// Nodes/Algebraic Container Ops/AddTo/Node_F_VN_AddToContainerElements_TcVnVector4_UINT
{attribute 'linkalways'} 
{attribute 'no_explicit_call' := 'This FB is a CLASS and must be accessed using methods or properties'}
{attribute 'enable_dynamic_creation'}
FUNCTION_BLOCK Node_F_VN_AddToContainerElements_TcVnVector4_UINT EXTENDS VisionNode
VAR
    aValue : _TcVnVector4_UINT;
    ipContainer : _ITcVnContainer;
    hrPrev : _HRESULT(S_OK);
    hresult : _HRESULT(S_OK);
END_VAR

METHOD FB_init : BOOL
VAR_INPUT
    bInitRetains : BOOL; // if TRUE, the retain variables are initialized (warm start / cold start)
    bInCopyCode : BOOL;  // if TRUE, the instance afterwards gets moved into the copy code (online change)
END_VAR
AddInput('aValue', aValue);
AddInput('ipContainer', ipContainer);
AddInput('hrPrev', hrPrev);
AddOutput('ipContainer', ipContainer);
AddOutput('hresult',hresult);
END_METHOD

METHOD PUBLIC  Clone : I_Node
VAR
    pNode : POINTER TO Node_F_VN_AddToContainerElements_TcVnVector4_UINT;
END_VAR
pNode := __NEW(Node_F_VN_AddToContainerElements_TcVnVector4_UINT);
Clone := pNode^;
END_METHOD

METHOD PROTECTED OnExecute
hresult.Value := F_VN_AddToContainerElements_TcVnVector4_UINT(
    aValue := aValue.Value,
    ipContainer := ipContainer.Value,
    hrPrev:= hrPrev.Value);
END_METHOD

METHOD PUBLIC PreExecutionCheck
VAR_INPUT
    Check : I_PreExecutionChecks;
END_VAR
Check.IsTrue(ipContainer.IsValid, 'ipContainer must be a valid container');
Check.IsTrue(ipContainer.IsType(TC_GLOBAL_CONST_LIST.ContainerType_Vector_TcVnVector4_UINT), 'ipContainer contains incorrect type');
END_METHOD

END_FUNCTION_BLOCK

// Nodes/Algebraic Container Ops/AddTo/Node_F_VN_AddToContainerElements_TcVnVector4_USINT
{attribute 'linkalways'} 
{attribute 'no_explicit_call' := 'This FB is a CLASS and must be accessed using methods or properties'}
{attribute 'enable_dynamic_creation'}
FUNCTION_BLOCK Node_F_VN_AddToContainerElements_TcVnVector4_USINT EXTENDS VisionNode
VAR
    aValue : _TcVnVector4_USINT;
    ipContainer : _ITcVnContainer;
    hrPrev : _HRESULT(S_OK);
    hresult : _HRESULT(S_OK);
END_VAR

METHOD FB_init : BOOL
VAR_INPUT
    bInitRetains : BOOL; // if TRUE, the retain variables are initialized (warm start / cold start)
    bInCopyCode : BOOL;  // if TRUE, the instance afterwards gets moved into the copy code (online change)
END_VAR
AddInput('aValue', aValue);
AddInput('ipContainer', ipContainer);
AddInput('hrPrev', hrPrev);
AddOutput('ipContainer', ipContainer);
AddOutput('hresult',hresult);
END_METHOD

METHOD PUBLIC  Clone : I_Node
VAR
    pNode : POINTER TO Node_F_VN_AddToContainerElements_TcVnVector4_USINT;
END_VAR
pNode := __NEW(Node_F_VN_AddToContainerElements_TcVnVector4_USINT);
Clone := pNode^;
END_METHOD

METHOD PROTECTED OnExecute
hresult.Value := F_VN_AddToContainerElements_TcVnVector4_USINT(
    aValue := aValue.Value,
    ipContainer := ipContainer.Value,
    hrPrev:= hrPrev.Value);
END_METHOD

METHOD PUBLIC PreExecutionCheck
VAR_INPUT
    Check : I_PreExecutionChecks;
END_VAR
Check.IsTrue(ipContainer.IsValid, 'ipContainer must be a valid container');
Check.IsTrue(ipContainer.IsType(TC_GLOBAL_CONST_LIST.ContainerType_Vector_TcVnVector4_USINT), 'ipContainer contains incorrect type');
END_METHOD

END_FUNCTION_BLOCK

// Nodes/Algebraic Container Ops/AddTo/Node_F_VN_AddToContainerElements_UDINT
{attribute 'linkalways'} 
{attribute 'no_explicit_call' := 'This FB is a CLASS and must be accessed using methods or properties'}
{attribute 'enable_dynamic_creation'}
FUNCTION_BLOCK Node_F_VN_AddToContainerElements_UDINT EXTENDS VisionNode
VAR
    nValue : _UDINT(0);
    ipContainer : _ITcVnContainer;
    hrPrev : _HRESULT(S_OK);
    hresult : _HRESULT(S_OK);
END_VAR

METHOD FB_init : BOOL
VAR_INPUT
    bInitRetains : BOOL; // if TRUE, the retain variables are initialized (warm start / cold start)
    bInCopyCode : BOOL;  // if TRUE, the instance afterwards gets moved into the copy code (online change)
END_VAR
AddParameter('nValue', nValue);
AddInput('ipContainer', ipContainer);
AddInput('hrPrev', hrPrev);
AddOutput('ipContainer', ipContainer);
AddOutput('hresult',hresult);
END_METHOD

METHOD PUBLIC  Clone : I_Node
VAR
    pNode : POINTER TO Node_F_VN_AddToContainerElements_UDINT;
END_VAR
pNode := __NEW(Node_F_VN_AddToContainerElements_UDINT);
Clone := pNode^;
END_METHOD

METHOD PROTECTED OnExecute
hresult.Value := F_VN_AddToContainerElements_UDINT(
    nValue := nValue.Value,
    ipContainer := ipContainer.Value,
    hrPrev:= hrPrev.Value);
END_METHOD

METHOD PUBLIC PreExecutionCheck
VAR_INPUT
    Check : I_PreExecutionChecks;
END_VAR
Check.IsTrue(ipContainer.IsValid, 'ipContainer must be a valid container');
Check.IsTrue(ipContainer.IsType(TC_GLOBAL_CONST_LIST.ContainerType_Vector_UDINT), 'ipContainer contains incorrect type');
END_METHOD

END_FUNCTION_BLOCK

// Nodes/Algebraic Container Ops/AddTo/Node_F_VN_AddToContainerElements_UINT
{attribute 'linkalways'} 
{attribute 'no_explicit_call' := 'This FB is a CLASS and must be accessed using methods or properties'}
{attribute 'enable_dynamic_creation'}
FUNCTION_BLOCK Node_F_VN_AddToContainerElements_UINT EXTENDS VisionNode
VAR
    nValue : _UINT(0);
    ipContainer : _ITcVnContainer;
    hrPrev : _HRESULT(S_OK);
    hresult : _HRESULT(S_OK);
END_VAR

METHOD FB_init : BOOL
VAR_INPUT
    bInitRetains : BOOL; // if TRUE, the retain variables are initialized (warm start / cold start)
    bInCopyCode : BOOL;  // if TRUE, the instance afterwards gets moved into the copy code (online change)
END_VAR
AddParameter('nValue', nValue);
AddInput('ipContainer', ipContainer);
AddInput('hrPrev', hrPrev);
AddOutput('ipContainer', ipContainer);
AddOutput('hresult',hresult);
END_METHOD

METHOD PUBLIC  Clone : I_Node
VAR
    pNode : POINTER TO Node_F_VN_AddToContainerElements_UINT;
END_VAR
pNode := __NEW(Node_F_VN_AddToContainerElements_UINT);
Clone := pNode^;
END_METHOD

METHOD PROTECTED OnExecute
hresult.Value := F_VN_AddToContainerElements_UINT(
    nValue := nValue.Value,
    ipContainer := ipContainer.Value,
    hrPrev:= hrPrev.Value);
END_METHOD

METHOD PUBLIC PreExecutionCheck
VAR_INPUT
    Check : I_PreExecutionChecks;
END_VAR
Check.IsTrue(ipContainer.IsValid, 'ipContainer must be a valid container');
Check.IsTrue(ipContainer.IsType(TC_GLOBAL_CONST_LIST.ContainerType_Vector_UINT), 'ipContainer contains incorrect type');
END_METHOD

END_FUNCTION_BLOCK

// Nodes/Algebraic Container Ops/AddTo/Node_F_VN_AddToContainerElements_ULINT
{attribute 'linkalways'} 
{attribute 'no_explicit_call' := 'This FB is a CLASS and must be accessed using methods or properties'}
{attribute 'enable_dynamic_creation'}
FUNCTION_BLOCK Node_F_VN_AddToContainerElements_ULINT EXTENDS VisionNode
VAR
    nValue : _ULINT(0);
    ipContainer : _ITcVnContainer;
    hrPrev : _HRESULT(S_OK);
    hresult : _HRESULT(S_OK);
END_VAR

METHOD FB_init : BOOL
VAR_INPUT
    bInitRetains : BOOL; // if TRUE, the retain variables are initialized (warm start / cold start)
    bInCopyCode : BOOL;  // if TRUE, the instance afterwards gets moved into the copy code (online change)
END_VAR
AddParameter('nValue', nValue);
AddInput('ipContainer', ipContainer);
AddInput('hrPrev', hrPrev);
AddOutput('ipContainer', ipContainer);
AddOutput('hresult',hresult);
END_METHOD

METHOD PUBLIC  Clone : I_Node
VAR
    pNode : POINTER TO Node_F_VN_AddToContainerElements_ULINT;
END_VAR
pNode := __NEW(Node_F_VN_AddToContainerElements_ULINT);
Clone := pNode^;
END_METHOD

METHOD PROTECTED OnExecute
hresult.Value := F_VN_AddToContainerElements_ULINT(
    nValue := nValue.Value,
    ipContainer := ipContainer.Value,
    hrPrev:= hrPrev.Value);
END_METHOD

METHOD PUBLIC PreExecutionCheck
VAR_INPUT
    Check : I_PreExecutionChecks;
END_VAR
Check.IsTrue(ipContainer.IsValid, 'ipContainer must be a valid container');
Check.IsTrue(ipContainer.IsType(TC_GLOBAL_CONST_LIST.ContainerType_Vector_ULINT), 'ipContainer contains incorrect type');
END_METHOD

END_FUNCTION_BLOCK

// Nodes/Algebraic Container Ops/AddTo/Node_F_VN_AddToContainerElements_USINT
{attribute 'linkalways'} 
{attribute 'no_explicit_call' := 'This FB is a CLASS and must be accessed using methods or properties'}
{attribute 'enable_dynamic_creation'}
FUNCTION_BLOCK Node_F_VN_AddToContainerElements_USINT EXTENDS VisionNode
VAR
    nValue : _USINT(0);
    ipContainer : _ITcVnContainer;
    hrPrev : _HRESULT(S_OK);
    hresult : _HRESULT(S_OK);
END_VAR

METHOD FB_init : BOOL
VAR_INPUT
    bInitRetains : BOOL; // if TRUE, the retain variables are initialized (warm start / cold start)
    bInCopyCode : BOOL;  // if TRUE, the instance afterwards gets moved into the copy code (online change)
END_VAR
AddParameter('nValue', nValue);
AddInput('ipContainer', ipContainer);
AddInput('hrPrev', hrPrev);
AddOutput('ipContainer', ipContainer);
AddOutput('hresult',hresult);
END_METHOD

METHOD PUBLIC  Clone : I_Node
VAR
    pNode : POINTER TO Node_F_VN_AddToContainerElements_USINT;
END_VAR
pNode := __NEW(Node_F_VN_AddToContainerElements_USINT);
Clone := pNode^;
END_METHOD

METHOD PROTECTED OnExecute
hresult.Value := F_VN_AddToContainerElements_USINT(
    nValue := nValue.Value,
    ipContainer := ipContainer.Value,
    hrPrev:= hrPrev.Value);
END_METHOD

METHOD PUBLIC PreExecutionCheck
VAR_INPUT
    Check : I_PreExecutionChecks;
END_VAR
Check.IsTrue(ipContainer.IsValid, 'ipContainer must be a valid container');
Check.IsTrue(ipContainer.IsType(TC_GLOBAL_CONST_LIST.ContainerType_Vector_USINT), 'ipContainer contains incorrect type');
END_METHOD

END_FUNCTION_BLOCK

// Nodes/Algebraic Container Ops/Node_F_VN_AddContainers
{attribute 'linkalways'} 
{attribute 'no_explicit_call' := 'This FB is a CLASS and must be accessed using methods or properties'}
{attribute 'enable_dynamic_creation'}
FUNCTION_BLOCK Node_F_VN_AddContainers EXTENDS VisionNode
VAR
    ipSrcContainer1 : _ITcVnContainer;
    ipSrcContainer2 : _ITcVnContainer;
    ipDestContainer : _ITcVnContainer;
    hrPrev : _HRESULT(S_OK);
    hresult : _HRESULT(S_OK);
END_VAR

METHOD FB_init : BOOL
VAR_INPUT
    bInitRetains : BOOL; // if TRUE, the retain variables are initialized (warm start / cold start)
    bInCopyCode : BOOL;  // if TRUE, the instance afterwards gets moved into the copy code (online change)
END_VAR
AddInput('ipSrcContainer1', ipSrcContainer1);
AddInput('ipSrcContainer2', ipSrcContainer2);
AddInput('hrPrev', hrPrev);
AddOutput('ipDestContainer', ipDestContainer);
AddOutput('hresult',hresult);
END_METHOD

METHOD PUBLIC  Clone : I_Node
VAR
    pNode : POINTER TO Node_F_VN_AddContainers;
END_VAR
pNode := __NEW(Node_F_VN_AddContainers);
Clone := pNode^;
END_METHOD

METHOD PROTECTED OnExecute
hresult.Value := F_VN_AddContainers(
    ipSrcContainer1 := ipSrcContainer1.Value,
    ipSrcContainer2 := ipSrcContainer2.Value,
    ipDestContainer := ipDestContainer.Value,
    hrPrev:= hrPrev.Value);
END_METHOD

METHOD PUBLIC PreExecutionCheck
VAR_INPUT
    Check : I_PreExecutionChecks;
END_VAR
Check.IsTrue(ipSrcContainer1.IsValid, 'ipSrcContainer1 must be a valid container');
Check.IsTrue(ipSrcContainer2.IsValid, 'ipSrcContainer2 must be a valid container');
Check.IsTrue(ContainersHaveMatchingTypes(ipSrcContainer1.Value, ipSrcContainer2.Value), 'Source containers must have matching types');
Check.IsTrue(ContainersHaveMatchingNumberOfElements(ipSrcContainer1.Value, ipSrcContainer2.Value), 'Source containers must contain the same number of elements');
END_METHOD

END_FUNCTION_BLOCK

// Nodes/Algebraic Container Ops/Node_F_VN_BitwiseAndContainers
{attribute 'linkalways'} 
{attribute 'no_explicit_call' := 'This FB is a CLASS and must be accessed using methods or properties'}
{attribute 'enable_dynamic_creation'}
FUNCTION_BLOCK Node_F_VN_BitwiseAndContainers EXTENDS VisionNode
VAR
    ipSrcContainer1 : _ITcVnContainer;
    ipSrcContainer2 : _ITcVnContainer;
    ipDestContainer : _ITcVnContainer;
    hrPrev : _HRESULT(S_OK);
    hresult : _HRESULT(S_OK);
END_VAR

METHOD FB_init : BOOL
VAR_INPUT
    bInitRetains : BOOL; // if TRUE, the retain variables are initialized (warm start / cold start)
    bInCopyCode : BOOL;  // if TRUE, the instance afterwards gets moved into the copy code (online change)
END_VAR
AddInput('ipSrcContainer1', ipSrcContainer1);
AddInput('ipSrcContainer2', ipSrcContainer2);
AddInput('hrPrev', hrPrev);
AddOutput('ipDestContainer', ipDestContainer);
AddOutput('hresult',hresult);
END_METHOD

METHOD PUBLIC  Clone : I_Node
VAR
    pNode : POINTER TO Node_F_VN_BitwiseAndContainers;
END_VAR
pNode := __NEW(Node_F_VN_BitwiseAndContainers);
Clone := pNode^;
END_METHOD

METHOD PROTECTED OnExecute
hresult.Value := F_VN_BitwiseAndContainers(
    ipSrcContainer1 := ipSrcContainer1.Value,
    ipSrcContainer2 := ipSrcContainer2.Value,
    ipDestContainer := ipDestContainer.Value,
    hrPrev:= hrPrev.Value);
END_METHOD

METHOD PUBLIC PreExecutionCheck
VAR_INPUT
    Check : I_PreExecutionChecks;
END_VAR
Check.IsTrue(ipSrcContainer1.IsValid, 'ipSrcContainer1 must be a valid container');
Check.IsTrue(ipSrcContainer2.IsValid, 'ipSrcContainer2 must be a valid container');
Check.IsTrue(ContainersHaveMatchingTypes(ipSrcContainer1.Value, ipSrcContainer2.Value), 'Source containers must have matching types');
Check.IsTrue(ContainersHaveMatchingNumberOfElements(ipSrcContainer1.Value, ipSrcContainer2.Value), 'Source containers must contain the same number of elements');


//TODO Need to check that container has integer values only.
// SINT, USINT, INT, UINT, DINT, UDINT, ULINT only?
END_METHOD

END_FUNCTION_BLOCK

// Nodes/Algebraic Container Ops/Node_F_VN_BitwiseNotContainer
{attribute 'linkalways'} 
{attribute 'no_explicit_call' := 'This FB is a CLASS and must be accessed using methods or properties'}
{attribute 'enable_dynamic_creation'}
FUNCTION_BLOCK Node_F_VN_BitwiseNotContainer EXTENDS VisionNode
VAR
    ipSrcContainer : _ITcVnContainer;
    ipDestContainer : _ITcVnContainer;
    hrPrev : _HRESULT(S_OK);
    hresult : _HRESULT(S_OK);
END_VAR

METHOD FB_init : BOOL
VAR_INPUT
    bInitRetains : BOOL; // if TRUE, the retain variables are initialized (warm start / cold start)
    bInCopyCode : BOOL;  // if TRUE, the instance afterwards gets moved into the copy code (online change)
END_VAR
AddInput('ipSrcContainer', ipSrcContainer);
AddInput('hrPrev', hrPrev);
AddOutput('ipDestContainer', ipDestContainer);
AddOutput('hresult',hresult);
END_METHOD

METHOD PUBLIC  Clone : I_Node
VAR
    pNode : POINTER TO Node_F_VN_BitwiseNotContainer;
END_VAR
pNode := __NEW(Node_F_VN_BitwiseNotContainer);
Clone := pNode^;
END_METHOD

METHOD PROTECTED OnExecute
hresult.Value := F_VN_BitwiseNotContainer(
    ipSrcContainer := ipSrcContainer.Value,
    ipDestContainer := ipDestContainer.Value,
    hrPrev:= hrPrev.Value);
END_METHOD

METHOD PUBLIC PreExecutionCheck
VAR_INPUT
    Check : I_PreExecutionChecks;
END_VAR
Check.IsTrue(ipSrcContainer.IsValid, 'ipSrcContainer must be a valid container');

IF Check.Failed THEN
    RETURN;
END_IF

//TODO Need to check that container has integer values only.
// SINT, USINT, INT, UINT, DINT, UDINT, ULINT only?
END_METHOD

END_FUNCTION_BLOCK

// Nodes/Algebraic Container Ops/Node_F_VN_BitwiseOrContainers
{attribute 'linkalways'} 
{attribute 'no_explicit_call' := 'This FB is a CLASS and must be accessed using methods or properties'}
{attribute 'enable_dynamic_creation'}
FUNCTION_BLOCK Node_F_VN_BitwiseOrContainers EXTENDS VisionNode
VAR
    ipSrcContainer1 : _ITcVnContainer;
    ipSrcContainer2 : _ITcVnContainer;
    ipDestContainer : _ITcVnContainer;
    hrPrev : _HRESULT(S_OK);
    hresult : _HRESULT(S_OK);
END_VAR

METHOD FB_init : BOOL
VAR_INPUT
    bInitRetains : BOOL; // if TRUE, the retain variables are initialized (warm start / cold start)
    bInCopyCode : BOOL;  // if TRUE, the instance afterwards gets moved into the copy code (online change)
END_VAR
AddInput('ipSrcContainer1', ipSrcContainer1);
AddInput('ipSrcContainer2', ipSrcContainer2);
AddInput('hrPrev', hrPrev);
AddOutput('ipDestContainer', ipDestContainer);
AddOutput('hresult',hresult);
END_METHOD

METHOD PUBLIC  Clone : I_Node
VAR
    pNode : POINTER TO Node_F_VN_BitwiseOrContainers;
END_VAR
pNode := __NEW(Node_F_VN_BitwiseOrContainers);
Clone := pNode^;
END_METHOD

METHOD PROTECTED OnExecute
hresult.Value := F_VN_BitwiseOrContainers(
    ipSrcContainer1 := ipSrcContainer1.Value,
    ipSrcContainer2 := ipSrcContainer2.Value,
    ipDestContainer := ipDestContainer.Value,
    hrPrev:= hrPrev.Value);
END_METHOD

METHOD PUBLIC PreExecutionCheck
VAR_INPUT
    Check : I_PreExecutionChecks;
END_VAR
Check.IsTrue(ipSrcContainer1.IsValid, 'ipSrcContainer1 must be a valid container');
Check.IsTrue(ipSrcContainer2.IsValid, 'ipSrcContainer2 must be a valid container');
Check.IsTrue(ContainersHaveMatchingTypes(ipSrcContainer1.Value, ipSrcContainer2.Value), 'Source containers must have matching types');
Check.IsTrue(ContainersHaveMatchingNumberOfElements(ipSrcContainer1.Value, ipSrcContainer2.Value), 'Source containers must contain the same number of elements');


//TODO Need to check that container has integer values only.
// SINT, USINT, INT, UINT, DINT, UDINT, ULINT only?
END_METHOD

END_FUNCTION_BLOCK

// Nodes/Algebraic Container Ops/Node_F_VN_BitwiseXorContainers
{attribute 'linkalways'} 
{attribute 'no_explicit_call' := 'This FB is a CLASS and must be accessed using methods or properties'}
{attribute 'enable_dynamic_creation'}
FUNCTION_BLOCK Node_F_VN_BitwiseXorContainers EXTENDS VisionNode
VAR
    ipSrcContainer1 : _ITcVnContainer;
    ipSrcContainer2 : _ITcVnContainer;
    ipDestContainer : _ITcVnContainer;
    hrPrev : _HRESULT(S_OK);
    hresult : _HRESULT(S_OK);
END_VAR

METHOD FB_init : BOOL
VAR_INPUT
    bInitRetains : BOOL; // if TRUE, the retain variables are initialized (warm start / cold start)
    bInCopyCode : BOOL;  // if TRUE, the instance afterwards gets moved into the copy code (online change)
END_VAR
AddInput('ipSrcContainer1', ipSrcContainer1);
AddInput('ipSrcContainer2', ipSrcContainer2);
AddInput('hrPrev', hrPrev);
AddOutput('ipDestContainer', ipDestContainer);
AddOutput('hresult',hresult);
END_METHOD

METHOD PUBLIC  Clone : I_Node
VAR
    pNode : POINTER TO Node_F_VN_BitwiseXorContainers;
END_VAR
pNode := __NEW(Node_F_VN_BitwiseXorContainers);
Clone := pNode^;
END_METHOD

METHOD PROTECTED OnExecute
hresult.Value := F_VN_BitwiseXorContainers(
    ipSrcContainer1 := ipSrcContainer1.Value,
    ipSrcContainer2 := ipSrcContainer2.Value,
    ipDestContainer := ipDestContainer.Value,
    hrPrev:= hrPrev.Value);
END_METHOD

METHOD PUBLIC PreExecutionCheck
VAR_INPUT
    Check : I_PreExecutionChecks;
END_VAR
Check.IsTrue(ipSrcContainer1.IsValid, 'ipSrcContainer1 must be a valid container');
Check.IsTrue(ipSrcContainer2.IsValid, 'ipSrcContainer2 must be a valid container');
Check.IsTrue(ContainersHaveMatchingTypes(ipSrcContainer1.Value, ipSrcContainer2.Value), 'Source containers must have matching types');
Check.IsTrue(ContainersHaveMatchingNumberOfElements(ipSrcContainer1.Value, ipSrcContainer2.Value), 'Source containers must contain the same number of elements');

//TODO Need to check that container has integer values only.
// SINT, USINT, INT, UINT, DINT, UDINT, ULINT only?
END_METHOD

END_FUNCTION_BLOCK

// Nodes/Algebraic Container Ops/Node_F_VN_DivideContainers
{attribute 'linkalways'} 
{attribute 'no_explicit_call' := 'This FB is a CLASS and must be accessed using methods or properties'}
{attribute 'enable_dynamic_creation'}
FUNCTION_BLOCK Node_F_VN_DivideContainers EXTENDS VisionNode
VAR
    ipSrcContainer1 : _ITcVnContainer;
    ipSrcContainer2 : _ITcVnContainer;
    ipDestContainer : _ITcVnContainer;
    hrPrev : _HRESULT(S_OK);
    hresult : _HRESULT(S_OK);
END_VAR

METHOD FB_init : BOOL
VAR_INPUT
    bInitRetains : BOOL; // if TRUE, the retain variables are initialized (warm start / cold start)
    bInCopyCode : BOOL;  // if TRUE, the instance afterwards gets moved into the copy code (online change)
END_VAR
AddInput('ipSrcContainer1', ipSrcContainer1);
AddInput('ipSrcContainer2', ipSrcContainer2);
AddInput('hrPrev', hrPrev);
AddOutput('ipDestContainer', ipDestContainer);
AddOutput('hresult',hresult);
END_METHOD

METHOD PUBLIC  Clone : I_Node
VAR
    pNode : POINTER TO Node_F_VN_DivideContainers;
END_VAR
pNode := __NEW(Node_F_VN_DivideContainers);
Clone := pNode^;
END_METHOD

METHOD PROTECTED OnExecute
hresult.Value := F_VN_DivideContainers(
    ipSrcContainer1 := ipSrcContainer1.Value,
    ipSrcContainer2 := ipSrcContainer2.Value,
    ipDestContainer := ipDestContainer.Value,
    hrPrev:= hrPrev.Value);
END_METHOD

METHOD PUBLIC PreExecutionCheck
VAR_INPUT
    Check : I_PreExecutionChecks;
END_VAR
Check.IsTrue(ipSrcContainer1.IsValid, 'ipSrcContainer1 must be a valid container');
Check.IsTrue(ipSrcContainer2.IsValid, 'ipSrcContainer2 must be a valid container');
Check.IsTrue(ContainersHaveMatchingTypes(ipSrcContainer1.Value, ipSrcContainer2.Value), 'Source containers must have matching types');
Check.IsTrue(ContainersHaveMatchingNumberOfElements(ipSrcContainer1.Value, ipSrcContainer2.Value), 'Source containers must contain the same number of elements');
END_METHOD

END_FUNCTION_BLOCK

// Nodes/Algebraic Container Ops/Node_F_VN_DivideContainersExp
{attribute 'linkalways'} 
{attribute 'no_explicit_call' := 'This FB is a CLASS and must be accessed using methods or properties'}
{attribute 'enable_dynamic_creation'}
FUNCTION_BLOCK Node_F_VN_DivideContainersExp EXTENDS VisionNode
VAR
    ipSrcContainer1 : _ITcVnContainer;
    ipSrcContainer2 : _ITcVnContainer;
    ipDestContainer : _ITcVnContainer;
    nIntDivideByZeroResult : _LINT(0);
    hrPrev : _HRESULT(S_OK);
    hresult : _HRESULT(S_OK);
END_VAR

METHOD FB_init : BOOL
VAR_INPUT
    bInitRetains : BOOL; // if TRUE, the retain variables are initialized (warm start / cold start)
    bInCopyCode : BOOL;  // if TRUE, the instance afterwards gets moved into the copy code (online change)
END_VAR
AddInput('ipSrcContainer1', ipSrcContainer1);
AddInput('ipSrcContainer2', ipSrcContainer2);
AddParameter('nIntDivideByZeroResult', nIntDivideByZeroResult);
AddInput('hrPrev', hrPrev);
AddOutput('ipDestContainer', ipDestContainer);
AddOutput('hresult',hresult);
END_METHOD

METHOD PUBLIC  Clone : I_Node
VAR
    pNode : POINTER TO Node_F_VN_DivideContainersExp;
END_VAR
pNode := __NEW(Node_F_VN_DivideContainersExp);
Clone := pNode^;
END_METHOD

METHOD PROTECTED OnExecute
hresult.Value := F_VN_DivideContainersExp(
    ipSrcContainer1 := ipSrcContainer1.Value,
    ipSrcContainer2 := ipSrcContainer2.Value,
    nIntDivideByZeroResult := nIntDivideByZeroResult.Value,
    ipDestContainer := ipDestContainer.Value,
    hrPrev:= hrPrev.Value);
END_METHOD

METHOD PUBLIC PreExecutionCheck
VAR_INPUT
    Check : I_PreExecutionChecks;
END_VAR
Check.IsTrue(ipSrcContainer1.IsValid, 'ipSrcContainer1 must be a valid container');
Check.IsTrue(ipSrcContainer2.IsValid, 'ipSrcContainer2 must be a valid container');
Check.IsTrue(ContainersHaveMatchingTypes(ipSrcContainer1.Value, ipSrcContainer2.Value), 'Source containers must have matching types');
Check.IsTrue(ContainersHaveMatchingNumberOfElements(ipSrcContainer1.Value, ipSrcContainer2.Value), 'Source containers must contain the same number of elements');
END_METHOD

END_FUNCTION_BLOCK

// Nodes/Algebraic Container Ops/Node_F_VN_MaxContainer
{attribute 'linkalways'} 
{attribute 'no_explicit_call' := 'This FB is a CLASS and must be accessed using methods or properties'}
{attribute 'enable_dynamic_creation'}
FUNCTION_BLOCK Node_F_VN_MaxContainer EXTENDS VisionNode
VAR
    ipSrcContainer1 : _ITcVnContainer;
    ipSrcContainer2 : _ITcVnContainer;
    ipDestContainer : _ITcVnContainer;
    hrPrev : _HRESULT(S_OK);
    hresult : _HRESULT(S_OK);
END_VAR

METHOD FB_init : BOOL
VAR_INPUT
    bInitRetains : BOOL; // if TRUE, the retain variables are initialized (warm start / cold start)
    bInCopyCode : BOOL;  // if TRUE, the instance afterwards gets moved into the copy code (online change)
END_VAR
AddInput('ipSrcContainer1', ipSrcContainer1);
AddInput('ipSrcContainer2', ipSrcContainer2);
AddInput('hrPrev', hrPrev);
AddOutput('ipDestContainer', ipDestContainer);
AddOutput('hresult',hresult);
END_METHOD

METHOD PUBLIC  Clone : I_Node
VAR
    pNode : POINTER TO Node_F_VN_MaxContainer;
END_VAR
pNode := __NEW(Node_F_VN_MaxContainer);
Clone := pNode^;
END_METHOD

METHOD PROTECTED OnExecute
hresult.Value := F_VN_MaxContainer(
    ipSrcContainer1 := ipSrcContainer1.Value,
    ipSrcContainer2 := ipSrcContainer2.Value,
    ipDestContainer := ipDestContainer.Value,
    hrPrev:= hrPrev.Value);
END_METHOD

METHOD PUBLIC PreExecutionCheck
VAR_INPUT
    Check : I_PreExecutionChecks;
END_VAR
Check.IsTrue(ipSrcContainer1.IsValid, 'ipSrcContainer1 must be a valid container');
Check.IsTrue(ipSrcContainer2.IsValid, 'ipSrcContainer2 must be a valid container');
Check.IsTrue(ContainersHaveMatchingTypes(ipSrcContainer1.Value, ipSrcContainer2.Value), 'Source containers must have matching types');
Check.IsTrue(ContainersHaveMatchingNumberOfElements(ipSrcContainer1.Value, ipSrcContainer2.Value), 'Source containers must contain the same number of elements');
END_METHOD

END_FUNCTION_BLOCK

// Nodes/Algebraic Container Ops/Node_F_VN_MinContainer
{attribute 'linkalways'} 
{attribute 'no_explicit_call' := 'This FB is a CLASS and must be accessed using methods or properties'}
{attribute 'enable_dynamic_creation'}
FUNCTION_BLOCK Node_F_VN_MinContainer EXTENDS VisionNode
VAR
    ipSrcContainer1 : _ITcVnContainer;
    ipSrcContainer2 : _ITcVnContainer;
    ipDestContainer : _ITcVnContainer;
    hrPrev : _HRESULT(S_OK);
    hresult : _HRESULT(S_OK);
END_VAR

METHOD FB_init : BOOL
VAR_INPUT
    bInitRetains : BOOL; // if TRUE, the retain variables are initialized (warm start / cold start)
    bInCopyCode : BOOL;  // if TRUE, the instance afterwards gets moved into the copy code (online change)
END_VAR
AddInput('ipSrcContainer1', ipSrcContainer1);
AddInput('ipSrcContainer2', ipSrcContainer2);
AddInput('hrPrev', hrPrev);
AddOutput('ipDestContainer', ipDestContainer);
AddOutput('hresult',hresult);
END_METHOD

METHOD PUBLIC  Clone : I_Node
VAR
    pNode : POINTER TO Node_F_VN_MinContainer;
END_VAR
pNode := __NEW(Node_F_VN_MinContainer);
Clone := pNode^;
END_METHOD

METHOD PROTECTED OnExecute
hresult.Value := F_VN_MinContainer(
    ipSrcContainer1 := ipSrcContainer1.Value,
    ipSrcContainer2 := ipSrcContainer2.Value,
    ipDestContainer := ipDestContainer.Value,
    hrPrev:= hrPrev.Value);
END_METHOD

METHOD PUBLIC PreExecutionCheck
VAR_INPUT
    Check : I_PreExecutionChecks;
END_VAR
Check.IsTrue(ipSrcContainer1.IsValid, 'ipSrcContainer1 must be a valid container');
Check.IsTrue(ipSrcContainer2.IsValid, 'ipSrcContainer2 must be a valid container');
Check.IsTrue(ContainersHaveMatchingTypes(ipSrcContainer1.Value, ipSrcContainer2.Value), 'Source containers must have matching types');
Check.IsTrue(ContainersHaveMatchingNumberOfElements(ipSrcContainer1.Value, ipSrcContainer2.Value), 'Source containers must contain the same number of elements');
END_METHOD

END_FUNCTION_BLOCK

// Nodes/Algebraic Container Ops/Node_F_VN_MultiplyContainers
{attribute 'linkalways'} 
{attribute 'no_explicit_call' := 'This FB is a CLASS and must be accessed using methods or properties'}
{attribute 'enable_dynamic_creation'}
FUNCTION_BLOCK Node_F_VN_MultiplyContainers EXTENDS VisionNode
VAR
    ipSrcContainer1 : _ITcVnContainer;
    ipSrcContainer2 : _ITcVnContainer;
    ipDestContainer : _ITcVnContainer;
    hrPrev : _HRESULT(S_OK);
    hresult : _HRESULT(S_OK);
END_VAR

METHOD FB_init : BOOL
VAR_INPUT
    bInitRetains : BOOL; // if TRUE, the retain variables are initialized (warm start / cold start)
    bInCopyCode : BOOL;  // if TRUE, the instance afterwards gets moved into the copy code (online change)
END_VAR
AddInput('ipSrcContainer1', ipSrcContainer1);
AddInput('ipSrcContainer2', ipSrcContainer2);
AddInput('hrPrev', hrPrev);
AddOutput('ipDestContainer', ipDestContainer);
AddOutput('hresult',hresult);
END_METHOD

METHOD PUBLIC  Clone : I_Node
VAR
    pNode : POINTER TO Node_F_VN_MultiplyContainers;
END_VAR
pNode := __NEW(Node_F_VN_MultiplyContainers);
Clone := pNode^;
END_METHOD

METHOD PROTECTED OnExecute
hresult.Value := F_VN_MultiplyContainers(
    ipSrcContainer1 := ipSrcContainer1.Value,
    ipSrcContainer2 := ipSrcContainer2.Value,
    ipDestContainer := ipDestContainer.Value,
    hrPrev:= hrPrev.Value);
END_METHOD

METHOD PUBLIC PreExecutionCheck
VAR_INPUT
    Check : I_PreExecutionChecks;
END_VAR
Check.IsTrue(ipSrcContainer1.IsValid, 'ipSrcContainer1 must be a valid container');
Check.IsTrue(ipSrcContainer2.IsValid, 'ipSrcContainer2 must be a valid container');
Check.IsTrue(ContainersHaveMatchingTypes(ipSrcContainer1.Value, ipSrcContainer2.Value), 'Source containers must have matching types');
Check.IsTrue(ContainersHaveMatchingNumberOfElements(ipSrcContainer1.Value, ipSrcContainer2.Value), 'Source containers must contain the same number of elements');
END_METHOD

END_FUNCTION_BLOCK

// Nodes/Algebraic Container Ops/Node_F_VN_NegateContainer
{attribute 'linkalways'} 
{attribute 'no_explicit_call' := 'This FB is a CLASS and must be accessed using methods or properties'}
{attribute 'enable_dynamic_creation'}
FUNCTION_BLOCK Node_F_VN_NegateContainer EXTENDS VisionNode
VAR
    ipSrcContainer : _ITcVnContainer;
    ipDestContainer : _ITcVnContainer;
    hrPrev : _HRESULT(S_OK);
    hresult : _HRESULT(S_OK);
END_VAR

METHOD FB_init : BOOL
VAR_INPUT
    bInitRetains : BOOL; // if TRUE, the retain variables are initialized (warm start / cold start)
    bInCopyCode : BOOL;  // if TRUE, the instance afterwards gets moved into the copy code (online change)
END_VAR
AddInput('ipSrcContainer', ipSrcContainer);
AddInput('hrPrev', hrPrev);
AddOutput('ipDestContainer', ipDestContainer);
AddOutput('hresult',hresult);
END_METHOD

METHOD PUBLIC  Clone : I_Node
VAR
    pNode : POINTER TO Node_F_VN_NegateContainer;
END_VAR
pNode := __NEW(Node_F_VN_NegateContainer);
Clone := pNode^;
END_METHOD

METHOD PROTECTED OnExecute
hresult.Value := F_VN_NegateContainer(
    ipSrcContainer := ipSrcContainer.Value,
    ipDestContainer := ipDestContainer.Value,
    hrPrev:= hrPrev.Value);
END_METHOD

METHOD PUBLIC PreExecutionCheck
VAR_INPUT
    Check : I_PreExecutionChecks;
END_VAR
Check.IsTrue(ipSrcContainer.IsValid, 'ipSrcContainer must be a valid container');
END_METHOD

END_FUNCTION_BLOCK

// Nodes/Algebraic Container Ops/Node_F_VN_SubtractContainers
{attribute 'linkalways'} 
{attribute 'no_explicit_call' := 'This FB is a CLASS and must be accessed using methods or properties'}
{attribute 'enable_dynamic_creation'}
FUNCTION_BLOCK Node_F_VN_SubtractContainers EXTENDS VisionNode
VAR
    ipSrcContainer1 : _ITcVnContainer;
    ipSrcContainer2 : _ITcVnContainer;
    ipDestContainer : _ITcVnContainer;
    hrPrev : _HRESULT(S_OK);
    hresult : _HRESULT(S_OK);
END_VAR

METHOD FB_init : BOOL
VAR_INPUT
    bInitRetains : BOOL; // if TRUE, the retain variables are initialized (warm start / cold start)
    bInCopyCode : BOOL;  // if TRUE, the instance afterwards gets moved into the copy code (online change)
END_VAR
AddInput('ipSrcContainer1', ipSrcContainer1);
AddInput('ipSrcContainer2', ipSrcContainer2);
AddInput('hrPrev', hrPrev);
AddOutput('ipDestContainer', ipDestContainer);
AddOutput('hresult',hresult);
END_METHOD

METHOD PUBLIC  Clone : I_Node
VAR
    pNode : POINTER TO Node_F_VN_SubtractContainers;
END_VAR
pNode := __NEW(Node_F_VN_SubtractContainers);
Clone := pNode^;
END_METHOD

METHOD PROTECTED OnExecute
hresult.Value := F_VN_SubtractContainers(
    ipSrcContainer1 := ipSrcContainer1.Value,
    ipSrcContainer2 := ipSrcContainer2.Value,
    ipDestContainer := ipDestContainer.Value,
    hrPrev:= hrPrev.Value);
END_METHOD

METHOD PUBLIC PreExecutionCheck
VAR_INPUT
    Check : I_PreExecutionChecks;
END_VAR
Check.IsTrue(ipSrcContainer1.IsValid, 'ipSrcContainer1 must be a valid container');
Check.IsTrue(ipSrcContainer2.IsValid, 'ipSrcContainer2 must be a valid container');
Check.IsTrue(ContainersHaveMatchingTypes(ipSrcContainer1.Value, ipSrcContainer2.Value), 'Source containers must have matching types');
Check.IsTrue(ContainersHaveMatchingNumberOfElements(ipSrcContainer1.Value, ipSrcContainer2.Value), 'Source containers must contain the same number of elements');
END_METHOD

END_FUNCTION_BLOCK

// Nodes/Algebraic Image Ops/Node_F_VN_AddImages
{attribute 'linkalways'} 
{attribute 'no_explicit_call' := 'This FB is a CLASS and must be accessed using methods or properties'}
{attribute 'enable_dynamic_creation'}
FUNCTION_BLOCK Node_F_VN_AddImages EXTENDS VisionNode
VAR
    ipSrcImage1 : _ITcVnImage;
    ipSrcImage2 : _ITcVnImage;
    ipDestImage : _ITcVnImage;
    hrPrev : _HRESULT(S_OK);
	hresult : _HRESULT(S_OK);
END_VAR

METHOD FB_init : BOOL
VAR_INPUT
	bInitRetains : BOOL; // if TRUE, the retain variables are initialized (warm start / cold start)
	bInCopyCode : BOOL;  // if TRUE, the instance afterwards gets moved into the copy code (online change)
END_VAR
AddInput('ipSrcImage1', ipSrcImage1);
AddInput('ipSrcImage2', ipSrcImage2);
AddInput('hrPrev', hrPrev);
AddOutput('ipDestImage', ipDestImage);
AddOutput('hresult',hresult);
END_METHOD

METHOD PUBLIC  Clone : I_Node
VAR
	pNode : POINTER TO Node_F_VN_AddImages;
END_VAR
pNode := __NEW(Node_F_VN_AddImages);
Clone := pNode^;
END_METHOD

METHOD PROTECTED OnExecute
hresult.Value := F_VN_AddImages(
    ipSrcImage1 := ipSrcImage1.Value,
    ipSrcImage2 := ipSrcImage2.Value,
	ipDestImage := ipDestImage.Value,
	hrPrev:= hrPrev.Value);
END_METHOD

METHOD PUBLIC PreExecutionCheck
VAR_INPUT
	Check : I_PreExecutionChecks;
END_VAR
Check.IsTrue(ipSrcImage1.IsValid, 'ipSrcImage1 must contain an image');
Check.IsTrue(ipSrcImage2.IsValid, 'ipSrcImage2 must contain an image');
Check.IsTrue(IsImage1SizeEqualToImage2Size(ipSrcImage1.Value, ipSrcImage2.Value), 'ipSrcImage1 must be the same size as ipSrcImage2');
END_METHOD

END_FUNCTION_BLOCK

// Nodes/Algebraic Image Ops/Node_F_VN_AddImagesWeighted
{attribute 'linkalways'} 
{attribute 'no_explicit_call' := 'This FB is a CLASS and must be accessed using methods or properties'}
{attribute 'enable_dynamic_creation'}
FUNCTION_BLOCK Node_F_VN_AddImagesWeighted EXTENDS VisionNode
VAR
    ipSrcImage1 : _ITcVnImage;
    ipSrcImage2 : _ITcVnImage;
    ipDestImage : _ITcVnImage;
    fWeight1 : _LREAL(0.0);
    fWeight2 : _LREAL(0.0);
    fDelta : _LREAL(0.0);
    hrPrev : _HRESULT(S_OK);
	hresult : _HRESULT(S_OK);
END_VAR

METHOD FB_init : BOOL
VAR_INPUT
	bInitRetains : BOOL; // if TRUE, the retain variables are initialized (warm start / cold start)
	bInCopyCode : BOOL;  // if TRUE, the instance afterwards gets moved into the copy code (online change)
END_VAR
AddInput('ipSrcImage1', ipSrcImage1);
AddInput('ipSrcImage2', ipSrcImage2);
AddParameter('fWeight1', fWeight1);
AddParameter('fWeight2', fWeight2);
AddParameter('fDelta', fDelta);
AddInput('hrPrev', hrPrev);
AddOutput('ipDestImage', ipDestImage);
AddOutput('hresult',hresult);
END_METHOD

METHOD PUBLIC  Clone : I_Node
VAR
	pNode : POINTER TO Node_F_VN_AddImagesWeighted;
END_VAR
pNode := __NEW(Node_F_VN_AddImagesWeighted);
Clone := pNode^;
END_METHOD

METHOD PROTECTED OnExecute
hresult.Value := F_VN_AddImagesWeighted(
    ipSrcImage1 := ipSrcImage1.Value,
    ipSrcImage2 := ipSrcImage2.Value,
	ipDestImage := ipDestImage.Value,
    fWeight1 := fWeight1.Value,
    fWeight2 := fWeight2.Value,
    fDelta := fDelta.Value,
	hrPrev:= hrPrev.Value);
END_METHOD

METHOD PUBLIC PreExecutionCheck
VAR_INPUT
	Check : I_PreExecutionChecks;
END_VAR
Check.IsTrue(ipSrcImage1.IsValid, 'ipSrcImage1 must contain an image');
Check.IsTrue(ipSrcImage2.IsValid, 'ipSrcImage2 must contain an image');
Check.IsTrue(IsImage1SizeEqualToImage2Size(ipSrcImage1.Value, ipSrcImage2.Value), 'ipSrcImage1 must be the same size as ipSrcImage2');
END_METHOD

END_FUNCTION_BLOCK

// Nodes/Algebraic Image Ops/Node_F_VN_AddImagesWeightedExp
{attribute 'linkalways'} 
{attribute 'no_explicit_call' := 'This FB is a CLASS and must be accessed using methods or properties'}
{attribute 'enable_dynamic_creation'}
FUNCTION_BLOCK Node_F_VN_AddImagesWeightedExp EXTENDS VisionNode
VAR
    ipSrcImage1 : _ITcVnImage;
    ipSrcImage2 : _ITcVnImage;
    ipDestImage : _ITcVnImage;
    fWeight1 : _LREAL(0.0);
    fWeight2 : _LREAL(0.0);
    fDelta : _LREAL(0.0);
    eDestType : _ETcVnElementType(ETcVnElementType.TCVN_ET_SAME_AS_SOURCE);
    hrPrev : _HRESULT(S_OK);
	hresult : _HRESULT(S_OK);
END_VAR

METHOD FB_init : BOOL
VAR_INPUT
	bInitRetains : BOOL; // if TRUE, the retain variables are initialized (warm start / cold start)
	bInCopyCode : BOOL;  // if TRUE, the instance afterwards gets moved into the copy code (online change)
END_VAR
AddInput('ipSrcImage1', ipSrcImage1);
AddInput('ipSrcImage2', ipSrcImage2);
AddParameter('fWeight1', fWeight1);
AddParameter('fWeight2', fWeight2);
AddParameter('fDelta', fDelta);
AddParameter('eDestType', eDestType);
AddInput('hrPrev', hrPrev);
AddOutput('ipDestImage', ipDestImage);
AddOutput('hresult',hresult);
END_METHOD

METHOD PUBLIC  Clone : I_Node
VAR
	pNode : POINTER TO Node_F_VN_AddImagesWeightedExp;
END_VAR
pNode := __NEW(Node_F_VN_AddImagesWeightedExp);
Clone := pNode^;
END_METHOD

METHOD PROTECTED OnExecute
hresult.Value := F_VN_AddImagesWeightedExp(
    ipSrcImage1 := ipSrcImage1.Value,
    ipSrcImage2 := ipSrcImage2.Value,
	ipDestImage := ipDestImage.Value,
    fWeight1 := fWeight1.Value,
    fWeight2 := fWeight2.Value,
    fDelta := fDelta.Value,
    eDestType := eDestType.Value,
	hrPrev:= hrPrev.Value);
END_METHOD

METHOD PUBLIC PreExecutionCheck
VAR_INPUT
	Check : I_PreExecutionChecks;
END_VAR
Check.IsTrue(ipSrcImage1.IsValid, 'ipSrcImage1 must contain an image');
Check.IsTrue(ipSrcImage2.IsValid, 'ipSrcImage2 must contain an image');
Check.IsTrue(IsImage1SizeEqualToImage2Size(ipSrcImage1.Value, ipSrcImage2.Value), 'ipSrcImage1 must be the same size as ipSrcImage2');
END_METHOD

END_FUNCTION_BLOCK

// Nodes/Algebraic Image Ops/Node_F_VN_AddScalarToImage
{attribute 'linkalways'} 
{attribute 'no_explicit_call' := 'This FB is a CLASS and must be accessed using methods or properties'}
{attribute 'enable_dynamic_creation'}
FUNCTION_BLOCK Node_F_VN_AddScalarToImage EXTENDS VisionNode
VAR
    fScalar : _LREAL(0.0);
    ipSrcImage : _ITcVnImage;
    ipDestImage : _ITcVnImage;
    hrPrev : _HRESULT(S_OK);
	hresult : _HRESULT(S_OK);
END_VAR

METHOD FB_init : BOOL
VAR_INPUT
	bInitRetains : BOOL; // if TRUE, the retain variables are initialized (warm start / cold start)
	bInCopyCode : BOOL;  // if TRUE, the instance afterwards gets moved into the copy code (online change)
END_VAR
AddParameter('fScalar', fScalar);
AddInput('ipSrcImage', ipSrcImage);
AddInput('hrPrev', hrPrev);
AddOutput('ipDestImage', ipDestImage);
AddOutput('hresult',hresult);
END_METHOD

METHOD PUBLIC  Clone : I_Node
VAR
	pNode : POINTER TO Node_F_VN_AddScalarToImage;
END_VAR
pNode := __NEW(Node_F_VN_AddScalarToImage);
Clone := pNode^;
END_METHOD

METHOD PROTECTED OnExecute
hresult.Value := F_VN_AddScalarToImage(
    fScalar := fScalar.Value,
    ipSrcImage := ipSrcImage.Value,
	ipDestImage := ipDestImage.Value,
	hrPrev:= hrPrev.Value);
END_METHOD

METHOD PUBLIC PreExecutionCheck
VAR_INPUT
	Check : I_PreExecutionChecks;
END_VAR
Check.IsTrue(ipSrcImage.IsValid, 'ipSrcImage must contain an image');
END_METHOD

END_FUNCTION_BLOCK

// Nodes/Algebraic Image Ops/Node_F_VN_AddVectorToImage
{attribute 'linkalways'} 
{attribute 'no_explicit_call' := 'This FB is a CLASS and must be accessed using methods or properties'}
{attribute 'enable_dynamic_creation'}
FUNCTION_BLOCK Node_F_VN_AddVectorToImage EXTENDS VisionNode
VAR
    aVector : _TcVnVector4_LREAL;
    ipSrcImage : _ITcVnImage;
    ipDestImage : _ITcVnImage;
    hrPrev : _HRESULT(S_OK);
	hresult : _HRESULT(S_OK);
END_VAR

METHOD FB_init : BOOL
VAR_INPUT
	bInitRetains : BOOL; // if TRUE, the retain variables are initialized (warm start / cold start)
	bInCopyCode : BOOL;  // if TRUE, the instance afterwards gets moved into the copy code (online change)
END_VAR
AddInput('aVector', aVector);
AddInput('ipSrcImage', ipSrcImage);
AddInput('hrPrev', hrPrev);
AddOutput('ipDestImage', ipDestImage);
AddOutput('hresult',hresult);
END_METHOD

METHOD PUBLIC  Clone : I_Node
VAR
	pNode : POINTER TO Node_F_VN_AddVectorToImage;
END_VAR
pNode := __NEW(Node_F_VN_AddVectorToImage);
Clone := pNode^;
END_METHOD

METHOD PROTECTED OnExecute
hresult.Value := F_VN_AddVectorToImage(
    aVector := aVector.Value,
    ipSrcImage := ipSrcImage.Value,
	ipDestImage := ipDestImage.Value,
	hrPrev:= hrPrev.Value);
END_METHOD

METHOD PUBLIC PreExecutionCheck
VAR_INPUT
	Check : I_PreExecutionChecks;
END_VAR
Check.IsTrue(ipSrcImage.IsValid, 'ipSrcImage must contain an image');
END_METHOD

END_FUNCTION_BLOCK

// Nodes/Algebraic Image Ops/Node_F_VN_BitwiseAndImages
{attribute 'linkalways'} 
{attribute 'no_explicit_call' := 'This FB is a CLASS and must be accessed using methods or properties'}
{attribute 'enable_dynamic_creation'}
FUNCTION_BLOCK Node_F_VN_BitwiseAndImages EXTENDS VisionNode
VAR
    ipSrcImage1 : _ITcVnImage;
    ipSrcImage2 : _ITcVnImage;
    ipDestImage : _ITcVnImage;
    hrPrev : _HRESULT(S_OK);
	hresult : _HRESULT(S_OK);
END_VAR

METHOD FB_init : BOOL
VAR_INPUT
	bInitRetains : BOOL; // if TRUE, the retain variables are initialized (warm start / cold start)
	bInCopyCode : BOOL;  // if TRUE, the instance afterwards gets moved into the copy code (online change)
END_VAR
AddInput('ipSrcImage1', ipSrcImage1);
AddInput('ipSrcImage2', ipSrcImage2);
AddInput('hrPrev', hrPrev);
AddOutput('ipDestImage', ipDestImage);
AddOutput('hresult',hresult);
END_METHOD

METHOD PUBLIC  Clone : I_Node
VAR
	pNode : POINTER TO Node_F_VN_BitwiseAndImages;
END_VAR
pNode := __NEW(Node_F_VN_BitwiseAndImages);
Clone := pNode^;
END_METHOD

METHOD PROTECTED OnExecute
hresult.Value := F_VN_BitwiseAndImages(
    ipSrcImage1 := ipSrcImage1.Value,
    ipSrcImage2 := ipSrcImage2.Value,
	ipDestImage := ipDestImage.Value,
	hrPrev:= hrPrev.Value);
END_METHOD

METHOD PUBLIC PreExecutionCheck
VAR_INPUT
	Check : I_PreExecutionChecks;
END_VAR
Check.IsTrue(ipSrcImage1.IsValid, 'ipSrcImage1 must contain an image');
Check.IsTrue(ipSrcImage2.IsValid, 'ipSrcImage2 must contain an image');
Check.IsTrue(IsImage1SizeEqualToImage2Size(ipSrcImage1.Value, ipSrcImage2.Value), 'ipSrcImage1 must be the same size as ipSrcImage2');
END_METHOD

END_FUNCTION_BLOCK

// Nodes/Algebraic Image Ops/Node_F_VN_BitwiseAndImagesExp
{attribute 'linkalways'} 
{attribute 'no_explicit_call' := 'This FB is a CLASS and must be accessed using methods or properties'}
{attribute 'enable_dynamic_creation'}
FUNCTION_BLOCK Node_F_VN_BitwiseAndImagesExp EXTENDS VisionNode
VAR
    ipSrcImage1 : _ITcVnImage;
    ipSrcImage2 : _ITcVnImage;
    ipDestImage : _ITcVnImage;
    ipMask : _ITcVnImage;
    hrPrev : _HRESULT(S_OK);
	hresult : _HRESULT(S_OK);
END_VAR

METHOD FB_init : BOOL
VAR_INPUT
	bInitRetains : BOOL; // if TRUE, the retain variables are initialized (warm start / cold start)
	bInCopyCode : BOOL;  // if TRUE, the instance afterwards gets moved into the copy code (online change)
END_VAR
AddInput('ipSrcImage1', ipSrcImage1);
AddInput('ipSrcImage2', ipSrcImage2);
AddInput('ipMask', ipMask);
AddInput('hrPrev', hrPrev);
AddOutput('ipDestImage', ipDestImage);
AddOutput('hresult',hresult);
END_METHOD

METHOD PUBLIC  Clone : I_Node
VAR
	pNode : POINTER TO Node_F_VN_BitwiseAndImagesExp;
END_VAR
pNode := __NEW(Node_F_VN_BitwiseAndImagesExp);
Clone := pNode^;
END_METHOD

METHOD PROTECTED OnExecute
hresult.Value := F_VN_BitwiseAndImagesExp(
    ipSrcImage1 := ipSrcImage1.Value,
    ipSrcImage2 := ipSrcImage2.Value,
	ipDestImage := ipDestImage.Value,
    ipMask := ipMask.Value,
	hrPrev:= hrPrev.Value);
END_METHOD

METHOD PUBLIC PreExecutionCheck
VAR_INPUT
	Check : I_PreExecutionChecks;
END_VAR
Check.IsTrue(ipSrcImage1.IsValid, 'ipSrcImage1 must contain an image');
Check.IsTrue(ipSrcImage2.IsValid, 'ipSrcImage2 must contain an image');
Check.IsTrue(IsImage1SizeEqualToImage2Size(ipSrcImage1.Value, ipSrcImage2.Value), 'ipSrcImage1 must be the same size as ipSrcImage2');
Check.IsTrue(ipMask.IsValid, 'ipMask must contain an image');
Check.IsTrue(ipMask.HasChannelCount(1), 'ipMask must have 1 channel');
Check.IsTrue(ipMask.IsPixelDepth(8), 'ipMask must have 8 bit pixel depth');
Check.IsTrue(IsImage1SizeEqualToImage2Size(ipMask.Value, ipSrcImage1.Value), 'ipMask must be the same size as ipSrcImage1');
END_METHOD

END_FUNCTION_BLOCK

// Nodes/Algebraic Image Ops/Node_F_VN_BitwiseAndScalarWithImage
{attribute 'linkalways'} 
{attribute 'no_explicit_call' := 'This FB is a CLASS and must be accessed using methods or properties'}
{attribute 'enable_dynamic_creation'}
FUNCTION_BLOCK Node_F_VN_BitwiseAndScalarWithImage EXTENDS VisionNode
VAR
    fScalar : _LREAL(0.0);
    ipSrcImage : _ITcVnImage;
    ipDestImage : _ITcVnImage;
    hrPrev : _HRESULT(S_OK);
	hresult : _HRESULT(S_OK);
END_VAR

METHOD FB_init : BOOL
VAR_INPUT
	bInitRetains : BOOL; // if TRUE, the retain variables are initialized (warm start / cold start)
	bInCopyCode : BOOL;  // if TRUE, the instance afterwards gets moved into the copy code (online change)
END_VAR
AddParameter('fScalar', fScalar);
AddInput('ipSrcImage', ipSrcImage);
AddInput('hrPrev', hrPrev);
AddOutput('ipDestImage', ipDestImage);
AddOutput('hresult',hresult);
END_METHOD

METHOD PUBLIC  Clone : I_Node
VAR
	pNode : POINTER TO Node_F_VN_BitwiseAndScalarWithImage;
END_VAR
pNode := __NEW(Node_F_VN_BitwiseAndScalarWithImage);
Clone := pNode^;
END_METHOD

METHOD PROTECTED OnExecute
hresult.Value := F_VN_BitwiseAndScalarWithImage(
    fScalar := fScalar.Value,
    ipSrcImage := ipSrcImage.Value,
	ipDestImage := ipDestImage.Value,
	hrPrev:= hrPrev.Value);
END_METHOD

METHOD PUBLIC PreExecutionCheck
VAR_INPUT
	Check : I_PreExecutionChecks;
END_VAR
Check.IsTrue(ipSrcImage.IsValid, 'ipSrcImage must contain an image');
END_METHOD

END_FUNCTION_BLOCK

// Nodes/Algebraic Image Ops/Node_F_VN_BitwiseAndVectorWithImage
{attribute 'linkalways'} 
{attribute 'no_explicit_call' := 'This FB is a CLASS and must be accessed using methods or properties'}
{attribute 'enable_dynamic_creation'}
FUNCTION_BLOCK Node_F_VN_BitwiseAndVectorWithImage EXTENDS VisionNode
VAR
    aVector : _TcVnVector4_LREAL;
    ipSrcImage : _ITcVnImage;
    ipDestImage : _ITcVnImage;
    hrPrev : _HRESULT(S_OK);
	hresult : _HRESULT(S_OK);
END_VAR

METHOD FB_init : BOOL
VAR_INPUT
	bInitRetains : BOOL; // if TRUE, the retain variables are initialized (warm start / cold start)
	bInCopyCode : BOOL;  // if TRUE, the instance afterwards gets moved into the copy code (online change)
END_VAR
AddInput('aVector', aVector);
AddInput('ipSrcImage', ipSrcImage);
AddInput('hrPrev', hrPrev);
AddOutput('ipDestImage', ipDestImage);
AddOutput('hresult',hresult);
END_METHOD

METHOD PUBLIC  Clone : I_Node
VAR
	pNode : POINTER TO Node_F_VN_BitwiseAndVectorWithImage;
END_VAR
pNode := __NEW(Node_F_VN_BitwiseAndVectorWithImage);
Clone := pNode^;
END_METHOD

METHOD PROTECTED OnExecute
hresult.Value := F_VN_BitwiseAndVectorWithImage(
    aVector := aVector.Value,
    ipSrcImage := ipSrcImage.Value,
	ipDestImage := ipDestImage.Value,
	hrPrev:= hrPrev.Value);
END_METHOD

METHOD PUBLIC PreExecutionCheck
VAR_INPUT
	Check : I_PreExecutionChecks;
END_VAR
Check.IsTrue(ipSrcImage.IsValid, 'ipSrcImage must contain an image');
END_METHOD

END_FUNCTION_BLOCK

// Nodes/Algebraic Image Ops/Node_F_VN_BitwiseNotImage
{attribute 'linkalways'} 
{attribute 'no_explicit_call' := 'This FB is a CLASS and must be accessed using methods or properties'}
{attribute 'enable_dynamic_creation'}
FUNCTION_BLOCK Node_F_VN_BitwiseNotImage EXTENDS VisionNode
VAR
    ipSrcImage : _ITcVnImage;
    ipDestImage : _ITcVnImage;
    hrPrev : _HRESULT(S_OK);
	hresult : _HRESULT(S_OK);
END_VAR

METHOD FB_init : BOOL
VAR_INPUT
	bInitRetains : BOOL; // if TRUE, the retain variables are initialized (warm start / cold start)
	bInCopyCode : BOOL;  // if TRUE, the instance afterwards gets moved into the copy code (online change)
END_VAR
AddInput('ipSrcImage', ipSrcImage);
AddInput('hrPrev', hrPrev);
AddOutput('ipDestImage', ipDestImage);
AddOutput('hresult',hresult);
END_METHOD

METHOD PUBLIC  Clone : I_Node
VAR
	pNode : POINTER TO Node_F_VN_BitwiseNotImage;
END_VAR
pNode := __NEW(Node_F_VN_BitwiseNotImage);
Clone := pNode^;
END_METHOD

METHOD PROTECTED OnExecute
hresult.Value := F_VN_BitwiseNotImage(
    ipSrcImage := ipSrcImage.Value,
	ipDestImage := ipDestImage.Value,
	hrPrev:= hrPrev.Value);
END_METHOD

METHOD PUBLIC PreExecutionCheck
VAR_INPUT
	Check : I_PreExecutionChecks;
END_VAR
Check.IsTrue(ipSrcImage.IsValid, 'ipSrcImage must contain an image');
END_METHOD

END_FUNCTION_BLOCK

// Nodes/Algebraic Image Ops/Node_F_VN_BitwiseNotImageExp
{attribute 'linkalways'} 
{attribute 'no_explicit_call' := 'This FB is a CLASS and must be accessed using methods or properties'}
{attribute 'enable_dynamic_creation'}
FUNCTION_BLOCK Node_F_VN_BitwiseNotImageExp EXTENDS VisionNode
VAR
    ipSrcImage : _ITcVnImage;
    ipDestImage : _ITcVnImage;
    ipMask : _ITcVnImage;
    hrPrev : _HRESULT(S_OK);
	hresult : _HRESULT(S_OK);
END_VAR

METHOD FB_init : BOOL
VAR_INPUT
	bInitRetains : BOOL; // if TRUE, the retain variables are initialized (warm start / cold start)
	bInCopyCode : BOOL;  // if TRUE, the instance afterwards gets moved into the copy code (online change)
END_VAR
AddInput('ipSrcImage', ipSrcImage);
AddInput('ipMask', ipMask);
AddInput('hrPrev', hrPrev);
AddOutput('ipDestImage', ipDestImage);
AddOutput('hresult',hresult);
END_METHOD

METHOD PUBLIC  Clone : I_Node
VAR
	pNode : POINTER TO Node_F_VN_BitwiseNotImageExp;
END_VAR
pNode := __NEW(Node_F_VN_BitwiseNotImageExp);
Clone := pNode^;
END_METHOD

METHOD PROTECTED OnExecute
hresult.Value := F_VN_BitwiseNotImageExp(
    ipSrcImage := ipSrcImage.Value,
	ipDestImage := ipDestImage.Value,
    ipMask := ipMask.Value,
	hrPrev:= hrPrev.Value);
END_METHOD

METHOD PUBLIC PreExecutionCheck
VAR_INPUT
	Check : I_PreExecutionChecks;
END_VAR
Check.IsTrue(ipSrcImage.IsValid, 'ipSrcImage must contain an image');
Check.IsTrue(ipMask.IsValid, 'ipMask must contain an image');
Check.IsTrue(ipMask.HasChannelCount(1), 'ipMask must have 1 channel');
Check.IsTrue(ipMask.IsPixelDepth(8), 'ipMask must have 8 bit pixel depth');
Check.IsTrue(IsImage1SizeEqualToImage2Size(ipMask.Value, ipSrcImage.Value), 'ipMask must be the same size as ipSrcImage');
END_METHOD

END_FUNCTION_BLOCK

// Nodes/Algebraic Image Ops/Node_F_VN_BitwiseOrImages
{attribute 'linkalways'} 
{attribute 'no_explicit_call' := 'This FB is a CLASS and must be accessed using methods or properties'}
{attribute 'enable_dynamic_creation'}
FUNCTION_BLOCK Node_F_VN_BitwiseOrImages EXTENDS VisionNode
VAR
    ipSrcImage1 : _ITcVnImage;
    ipSrcImage2 : _ITcVnImage;
    ipDestImage : _ITcVnImage;
    hrPrev : _HRESULT(S_OK);
	hresult : _HRESULT(S_OK);
END_VAR

METHOD FB_init : BOOL
VAR_INPUT
	bInitRetains : BOOL; // if TRUE, the retain variables are initialized (warm start / cold start)
	bInCopyCode : BOOL;  // if TRUE, the instance afterwards gets moved into the copy code (online change)
END_VAR
AddInput('ipSrcImage1', ipSrcImage1);
AddInput('ipSrcImage2', ipSrcImage2);
AddInput('hrPrev', hrPrev);
AddOutput('ipDestImage', ipDestImage);
AddOutput('hresult',hresult);
END_METHOD

METHOD PUBLIC  Clone : I_Node
VAR
	pNode : POINTER TO Node_F_VN_BitwiseOrImages;
END_VAR
pNode := __NEW(Node_F_VN_BitwiseOrImages);
Clone := pNode^;
END_METHOD

METHOD PROTECTED OnExecute
hresult.Value := F_VN_BitwiseOrImages(
    ipSrcImage1 := ipSrcImage1.Value,
    ipSrcImage2 := ipSrcImage2.Value,
	ipDestImage := ipDestImage.Value,
	hrPrev:= hrPrev.Value);
END_METHOD

METHOD PUBLIC PreExecutionCheck
VAR_INPUT
	Check : I_PreExecutionChecks;
END_VAR
Check.IsTrue(ipSrcImage1.IsValid, 'ipSrcImage1 must contain an image');
Check.IsTrue(ipSrcImage2.IsValid, 'ipSrcImage2 must contain an image');
Check.IsTrue(IsImage1SizeEqualToImage2Size(ipSrcImage1.Value, ipSrcImage2.Value), 'ipSrcImage1 must be the same size as ipSrcImage2');
END_METHOD

END_FUNCTION_BLOCK

// Nodes/Algebraic Image Ops/Node_F_VN_BitwiseOrImagesExp
{attribute 'linkalways'} 
{attribute 'no_explicit_call' := 'This FB is a CLASS and must be accessed using methods or properties'}
{attribute 'enable_dynamic_creation'}
FUNCTION_BLOCK Node_F_VN_BitwiseOrImagesExp EXTENDS VisionNode
VAR
    ipSrcImage1 : _ITcVnImage;
    ipSrcImage2 : _ITcVnImage;
    ipDestImage : _ITcVnImage;
    ipMask : _ITcVnImage;
    hrPrev : _HRESULT(S_OK);
	hresult : _HRESULT(S_OK);
END_VAR

METHOD FB_init : BOOL
VAR_INPUT
	bInitRetains : BOOL; // if TRUE, the retain variables are initialized (warm start / cold start)
	bInCopyCode : BOOL;  // if TRUE, the instance afterwards gets moved into the copy code (online change)
END_VAR
AddInput('ipSrcImage1', ipSrcImage1);
AddInput('ipSrcImage2', ipSrcImage2);
AddInput('ipMask', ipMask);
AddInput('hrPrev', hrPrev);
AddOutput('ipDestImage', ipDestImage);
AddOutput('hresult',hresult);
END_METHOD

METHOD PUBLIC  Clone : I_Node
VAR
	pNode : POINTER TO Node_F_VN_BitwiseOrImagesExp;
END_VAR
pNode := __NEW(Node_F_VN_BitwiseOrImagesExp);
Clone := pNode^;
END_METHOD

METHOD PROTECTED OnExecute
hresult.Value := F_VN_BitwiseOrImagesExp(
    ipSrcImage1 := ipSrcImage1.Value,
    ipSrcImage2 := ipSrcImage2.Value,
	ipDestImage := ipDestImage.Value,
    ipMask := ipMask.Value,
	hrPrev:= hrPrev.Value);
END_METHOD

METHOD PUBLIC PreExecutionCheck
VAR_INPUT
	Check : I_PreExecutionChecks;
END_VAR
Check.IsTrue(ipSrcImage1.IsValid, 'ipSrcImage1 must contain an image');
Check.IsTrue(ipSrcImage2.IsValid, 'ipSrcImage2 must contain an image');
Check.IsTrue(IsImage1SizeEqualToImage2Size(ipSrcImage1.Value, ipSrcImage2.Value), 'ipSrcImage1 must be the same size as ipSrcImage2');
Check.IsTrue(ipMask.IsValid, 'ipMask must contain an image');
Check.IsTrue(ipMask.HasChannelCount(1), 'ipMask must have 1 channel');
Check.IsTrue(ipMask.IsPixelDepth(8), 'ipMask must have 8 bit pixel depth');
Check.IsTrue(IsImage1SizeEqualToImage2Size(ipMask.Value, ipSrcImage1.Value), 'ipMask must be the same size as ipSrcImage1');
END_METHOD

END_FUNCTION_BLOCK

// Nodes/Algebraic Image Ops/Node_F_VN_BitwiseOrScalarWithImage
{attribute 'linkalways'} 
{attribute 'no_explicit_call' := 'This FB is a CLASS and must be accessed using methods or properties'}
{attribute 'enable_dynamic_creation'}
FUNCTION_BLOCK Node_F_VN_BitwiseOrScalarWithImage EXTENDS VisionNode
VAR
    fScalar : _LREAL(0.0);
    ipSrcImage : _ITcVnImage;
    ipDestImage : _ITcVnImage;
    hrPrev : _HRESULT(S_OK);
	hresult : _HRESULT(S_OK);
END_VAR

METHOD FB_init : BOOL
VAR_INPUT
	bInitRetains : BOOL; // if TRUE, the retain variables are initialized (warm start / cold start)
	bInCopyCode : BOOL;  // if TRUE, the instance afterwards gets moved into the copy code (online change)
END_VAR
AddParameter('fScalar', fScalar);
AddInput('ipSrcImage', ipSrcImage);
AddInput('hrPrev', hrPrev);
AddOutput('ipDestImage', ipDestImage);
AddOutput('hresult',hresult);
END_METHOD

METHOD PUBLIC  Clone : I_Node
VAR
	pNode : POINTER TO Node_F_VN_BitwiseOrScalarWithImage;
END_VAR
pNode := __NEW(Node_F_VN_BitwiseOrScalarWithImage);
Clone := pNode^;
END_METHOD

METHOD PROTECTED OnExecute
hresult.Value := F_VN_BitwiseOrScalarWithImage(
    fScalar := fScalar.Value,
    ipSrcImage := ipSrcImage.Value,
	ipDestImage := ipDestImage.Value,
	hrPrev:= hrPrev.Value);
END_METHOD

METHOD PUBLIC PreExecutionCheck
VAR_INPUT
	Check : I_PreExecutionChecks;
END_VAR
Check.IsTrue(ipSrcImage.IsValid, 'ipSrcImage must contain an image');
END_METHOD

END_FUNCTION_BLOCK

// Nodes/Algebraic Image Ops/Node_F_VN_BitwiseOrVectorWithImage
{attribute 'linkalways'} 
{attribute 'no_explicit_call' := 'This FB is a CLASS and must be accessed using methods or properties'}
{attribute 'enable_dynamic_creation'}
FUNCTION_BLOCK Node_F_VN_BitwiseOrVectorWithImage EXTENDS VisionNode
VAR
    aVector : _TcVnVector4_LREAL;
    ipSrcImage : _ITcVnImage;
    ipDestImage : _ITcVnImage;
    hrPrev : _HRESULT(S_OK);
	hresult : _HRESULT(S_OK);
END_VAR

METHOD FB_init : BOOL
VAR_INPUT
	bInitRetains : BOOL; // if TRUE, the retain variables are initialized (warm start / cold start)
	bInCopyCode : BOOL;  // if TRUE, the instance afterwards gets moved into the copy code (online change)
END_VAR
AddInput('aVector', aVector);
AddInput('ipSrcImage', ipSrcImage);
AddInput('hrPrev', hrPrev);
AddOutput('ipDestImage', ipDestImage);
AddOutput('hresult',hresult);
END_METHOD

METHOD PUBLIC  Clone : I_Node
VAR
	pNode : POINTER TO Node_F_VN_BitwiseOrVectorWithImage;
END_VAR
pNode := __NEW(Node_F_VN_BitwiseOrVectorWithImage);
Clone := pNode^;
END_METHOD

METHOD PROTECTED OnExecute
hresult.Value := F_VN_BitwiseOrVectorWithImage(
    aVector := aVector.Value,
    ipSrcImage := ipSrcImage.Value,
	ipDestImage := ipDestImage.Value,
	hrPrev:= hrPrev.Value);
END_METHOD

METHOD PUBLIC PreExecutionCheck
VAR_INPUT
	Check : I_PreExecutionChecks;
END_VAR
Check.IsTrue(ipSrcImage.IsValid, 'ipSrcImage must contain an image');
END_METHOD

END_FUNCTION_BLOCK

// Nodes/Algebraic Image Ops/Node_F_VN_BitwiseXorImages
{attribute 'linkalways'} 
{attribute 'no_explicit_call' := 'This FB is a CLASS and must be accessed using methods or properties'}
{attribute 'enable_dynamic_creation'}
FUNCTION_BLOCK Node_F_VN_BitwiseXorImages EXTENDS VisionNode
VAR
    ipSrcImage1 : _ITcVnImage;
    ipSrcImage2 : _ITcVnImage;
    ipDestImage : _ITcVnImage;
    hrPrev : _HRESULT(S_OK);
	hresult : _HRESULT(S_OK);
END_VAR

METHOD FB_init : BOOL
VAR_INPUT
	bInitRetains : BOOL; // if TRUE, the retain variables are initialized (warm start / cold start)
	bInCopyCode : BOOL;  // if TRUE, the instance afterwards gets moved into the copy code (online change)
END_VAR
AddInput('ipSrcImage1', ipSrcImage1);
AddInput('ipSrcImage2', ipSrcImage2);
AddInput('hrPrev', hrPrev);
AddOutput('ipDestImage', ipDestImage);
AddOutput('hresult',hresult);
END_METHOD

METHOD PUBLIC  Clone : I_Node
VAR
	pNode : POINTER TO Node_F_VN_BitwiseXorImages;
END_VAR
pNode := __NEW(Node_F_VN_BitwiseXorImages);
Clone := pNode^;
END_METHOD

METHOD PROTECTED OnExecute
hresult.Value := F_VN_BitwiseXorImages(
    ipSrcImage1 := ipSrcImage1.Value,
    ipSrcImage2 := ipSrcImage2.Value,
	ipDestImage := ipDestImage.Value,
	hrPrev:= hrPrev.Value);
END_METHOD

METHOD PUBLIC PreExecutionCheck
VAR_INPUT
	Check : I_PreExecutionChecks;
END_VAR
Check.IsTrue(ipSrcImage1.IsValid, 'ipSrcImage1 must contain an image');
Check.IsTrue(ipSrcImage2.IsValid, 'ipSrcImage2 must contain an image');
Check.IsTrue(IsImage1SizeEqualToImage2Size(ipSrcImage1.Value, ipSrcImage2.Value), 'ipSrcImage1 must be the same size as ipSrcImage2');
END_METHOD

END_FUNCTION_BLOCK

// Nodes/Algebraic Image Ops/Node_F_VN_BitwiseXorImagesExp
{attribute 'linkalways'} 
{attribute 'no_explicit_call' := 'This FB is a CLASS and must be accessed using methods or properties'}
{attribute 'enable_dynamic_creation'}
FUNCTION_BLOCK Node_F_VN_BitwiseXorImagesExp EXTENDS VisionNode
VAR
    ipSrcImage1 : _ITcVnImage;
    ipSrcImage2 : _ITcVnImage;
    ipDestImage : _ITcVnImage;
    ipMask : _ITcVnImage;
    hrPrev : _HRESULT(S_OK);
	hresult : _HRESULT(S_OK);
END_VAR

METHOD FB_init : BOOL
VAR_INPUT
	bInitRetains : BOOL; // if TRUE, the retain variables are initialized (warm start / cold start)
	bInCopyCode : BOOL;  // if TRUE, the instance afterwards gets moved into the copy code (online change)
END_VAR
AddInput('ipSrcImage1', ipSrcImage1);
AddInput('ipSrcImage2', ipSrcImage2);
AddInput('ipMask', ipMask);
AddInput('hrPrev', hrPrev);
AddOutput('ipDestImage', ipDestImage);
AddOutput('hresult',hresult);
END_METHOD

METHOD PUBLIC  Clone : I_Node
VAR
	pNode : POINTER TO Node_F_VN_BitwiseXorImagesExp;
END_VAR
pNode := __NEW(Node_F_VN_BitwiseXorImagesExp);
Clone := pNode^;
END_METHOD

METHOD PROTECTED OnExecute
hresult.Value := F_VN_BitwiseXorImagesExp(
    ipSrcImage1 := ipSrcImage1.Value,
    ipSrcImage2 := ipSrcImage2.Value,
	ipDestImage := ipDestImage.Value,
    ipMask := ipMask.Value,
	hrPrev:= hrPrev.Value);
END_METHOD

METHOD PUBLIC PreExecutionCheck
VAR_INPUT
	Check : I_PreExecutionChecks;
END_VAR
Check.IsTrue(ipSrcImage1.IsValid, 'ipSrcImage1 must contain an image');
Check.IsTrue(ipSrcImage2.IsValid, 'ipSrcImage2 must contain an image');
Check.IsTrue(IsImage1SizeEqualToImage2Size(ipSrcImage1.Value, ipSrcImage2.Value), 'ipSrcImage1 must be the same size as ipSrcImage2');
Check.IsTrue(ipMask.IsValid, 'ipMask must contain an image');
Check.IsTrue(ipMask.HasChannelCount(1), 'ipMask must have 1 channel');
Check.IsTrue(ipMask.IsPixelDepth(8), 'ipMask must have 8 bit pixel depth');
Check.IsTrue(IsImage1SizeEqualToImage2Size(ipMask.Value, ipSrcImage1.Value), 'ipMask must be the same size as ipSrcImage1');
END_METHOD

END_FUNCTION_BLOCK

// Nodes/Algebraic Image Ops/Node_F_VN_BitwiseXorScalarWithImage
{attribute 'linkalways'} 
{attribute 'no_explicit_call' := 'This FB is a CLASS and must be accessed using methods or properties'}
{attribute 'enable_dynamic_creation'}
FUNCTION_BLOCK Node_F_VN_BitwiseXorScalarWithImage EXTENDS VisionNode
VAR
    fScalar : _LREAL(0.0);
    ipSrcImage : _ITcVnImage;
    ipDestImage : _ITcVnImage;
    hrPrev : _HRESULT(S_OK);
	hresult : _HRESULT(S_OK);
END_VAR

METHOD FB_init : BOOL
VAR_INPUT
	bInitRetains : BOOL; // if TRUE, the retain variables are initialized (warm start / cold start)
	bInCopyCode : BOOL;  // if TRUE, the instance afterwards gets moved into the copy code (online change)
END_VAR
AddParameter('fScalar', fScalar);
AddInput('ipSrcImage', ipSrcImage);
AddInput('hrPrev', hrPrev);
AddOutput('ipDestImage', ipDestImage);
AddOutput('hresult',hresult);
END_METHOD

METHOD PUBLIC  Clone : I_Node
VAR
	pNode : POINTER TO Node_F_VN_BitwiseXorScalarWithImage;
END_VAR
pNode := __NEW(Node_F_VN_BitwiseXorScalarWithImage);
Clone := pNode^;
END_METHOD

METHOD PROTECTED OnExecute
hresult.Value := F_VN_BitwiseXorScalarWithImage(
    fScalar := fScalar.Value,
    ipSrcImage := ipSrcImage.Value,
	ipDestImage := ipDestImage.Value,
	hrPrev:= hrPrev.Value);
END_METHOD

METHOD PUBLIC PreExecutionCheck
VAR_INPUT
	Check : I_PreExecutionChecks;
END_VAR
Check.IsTrue(ipSrcImage.IsValid, 'ipSrcImage must contain an image');
END_METHOD

END_FUNCTION_BLOCK

// Nodes/Algebraic Image Ops/Node_F_VN_BitwiseXorVectorWithImage
{attribute 'linkalways'} 
{attribute 'no_explicit_call' := 'This FB is a CLASS and must be accessed using methods or properties'}
{attribute 'enable_dynamic_creation'}
FUNCTION_BLOCK Node_F_VN_BitwiseXorVectorWithImage EXTENDS VisionNode
VAR
    aVector : _TcVnVector4_LREAL;
    ipSrcImage : _ITcVnImage;
    ipDestImage : _ITcVnImage;
    hrPrev : _HRESULT(S_OK);
	hresult : _HRESULT(S_OK);
END_VAR

METHOD FB_init : BOOL
VAR_INPUT
	bInitRetains : BOOL; // if TRUE, the retain variables are initialized (warm start / cold start)
	bInCopyCode : BOOL;  // if TRUE, the instance afterwards gets moved into the copy code (online change)
END_VAR
AddInput('aVector', aVector);
AddInput('ipSrcImage', ipSrcImage);
AddInput('hrPrev', hrPrev);
AddOutput('ipDestImage', ipDestImage);
AddOutput('hresult',hresult);
END_METHOD

METHOD PUBLIC  Clone : I_Node
VAR
	pNode : POINTER TO Node_F_VN_BitwiseXorVectorWithImage;
END_VAR
pNode := __NEW(Node_F_VN_BitwiseXorVectorWithImage);
Clone := pNode^;
END_METHOD

METHOD PROTECTED OnExecute
hresult.Value := F_VN_BitwiseXorVectorWithImage(
    aVector := aVector.Value,
    ipSrcImage := ipSrcImage.Value,
	ipDestImage := ipDestImage.Value,
	hrPrev:= hrPrev.Value);
END_METHOD

METHOD PUBLIC PreExecutionCheck
VAR_INPUT
	Check : I_PreExecutionChecks;
END_VAR
Check.IsTrue(ipSrcImage.IsValid, 'ipSrcImage must contain an image');
END_METHOD

END_FUNCTION_BLOCK

// Nodes/Algebraic Image Ops/Node_F_VN_DivideImageByScalar
{attribute 'linkalways'} 
{attribute 'no_explicit_call' := 'This FB is a CLASS and must be accessed using methods or properties'}
{attribute 'enable_dynamic_creation'}
FUNCTION_BLOCK Node_F_VN_DivideImageByScalar EXTENDS VisionNode
VAR
    ipSrcImage : _ITcVnImage;
    fScalar : _LREAL(0.0);
    ipDestImage : _ITcVnImage;
    hrPrev : _HRESULT(S_OK);
	hresult : _HRESULT(S_OK);
END_VAR

METHOD FB_init : BOOL
VAR_INPUT
	bInitRetains : BOOL; // if TRUE, the retain variables are initialized (warm start / cold start)
	bInCopyCode : BOOL;  // if TRUE, the instance afterwards gets moved into the copy code (online change)
END_VAR
AddInput('ipSrcImage', ipSrcImage);
AddParameter('fScalar', fScalar);
AddInput('hrPrev', hrPrev);
AddOutput('ipDestImage', ipDestImage);
AddOutput('hresult',hresult);
END_METHOD

METHOD PUBLIC  Clone : I_Node
VAR
	pNode : POINTER TO Node_F_VN_DivideImageByScalar;
END_VAR
pNode := __NEW(Node_F_VN_DivideImageByScalar);
Clone := pNode^;
END_METHOD

METHOD PROTECTED OnExecute
hresult.Value := F_VN_DivideImageByScalar(
    ipSrcImage := ipSrcImage.Value,
    fScalar := fScalar.Value,
	ipDestImage := ipDestImage.Value,
	hrPrev:= hrPrev.Value);
END_METHOD

METHOD PUBLIC PreExecutionCheck
VAR_INPUT
	Check : I_PreExecutionChecks;
END_VAR
Check.IsTrue(ipSrcImage.IsValid, 'ipSrcImage must contain an image');
END_METHOD

END_FUNCTION_BLOCK

// Nodes/Algebraic Image Ops/Node_F_VN_DivideImageByVector
{attribute 'linkalways'} 
{attribute 'no_explicit_call' := 'This FB is a CLASS and must be accessed using methods or properties'}
{attribute 'enable_dynamic_creation'}
FUNCTION_BLOCK Node_F_VN_DivideImageByVector EXTENDS VisionNode
VAR
    ipSrcImage : _ITcVnImage;
    aVector : _TcVnVector4_LREAL;
    ipDestImage : _ITcVnImage;
    hrPrev : _HRESULT(S_OK);
	hresult : _HRESULT(S_OK);
END_VAR

METHOD FB_init : BOOL
VAR_INPUT
	bInitRetains : BOOL; // if TRUE, the retain variables are initialized (warm start / cold start)
	bInCopyCode : BOOL;  // if TRUE, the instance afterwards gets moved into the copy code (online change)
END_VAR
AddInput('ipSrcImage', ipSrcImage);
AddInput('aVector', aVector);
AddInput('hrPrev', hrPrev);
AddOutput('ipDestImage', ipDestImage);
AddOutput('hresult',hresult);
END_METHOD

METHOD PUBLIC  Clone : I_Node
VAR
	pNode : POINTER TO Node_F_VN_DivideImageByVector;
END_VAR
pNode := __NEW(Node_F_VN_DivideImageByVector);
Clone := pNode^;
END_METHOD

METHOD PROTECTED OnExecute
hresult.Value := F_VN_DivideImageByVector(
    ipSrcImage := ipSrcImage.Value,
    aVector := aVector.Value,
	ipDestImage := ipDestImage.Value,
	hrPrev:= hrPrev.Value);
END_METHOD

METHOD PUBLIC PreExecutionCheck
VAR_INPUT
	Check : I_PreExecutionChecks;
END_VAR
Check.IsTrue(ipSrcImage.IsValid, 'ipSrcImage must contain an image');
END_METHOD

END_FUNCTION_BLOCK

// Nodes/Algebraic Image Ops/Node_F_VN_DivideImages
{attribute 'linkalways'} 
{attribute 'no_explicit_call' := 'This FB is a CLASS and must be accessed using methods or properties'}
{attribute 'enable_dynamic_creation'}
FUNCTION_BLOCK Node_F_VN_DivideImages EXTENDS VisionNode
VAR
    ipSrcImage1 : _ITcVnImage;
    ipSrcImage2 : _ITcVnImage;
    ipDestImage : _ITcVnImage;
    hrPrev : _HRESULT(S_OK);
	hresult : _HRESULT(S_OK);
END_VAR

METHOD FB_init : BOOL
VAR_INPUT
	bInitRetains : BOOL; // if TRUE, the retain variables are initialized (warm start / cold start)
	bInCopyCode : BOOL;  // if TRUE, the instance afterwards gets moved into the copy code (online change)
END_VAR
AddInput('ipSrcImage1', ipSrcImage1);
AddInput('ipSrcImage2', ipSrcImage2);
AddInput('hrPrev', hrPrev);
AddOutput('ipDestImage', ipDestImage);
AddOutput('hresult',hresult);
END_METHOD

METHOD PUBLIC  Clone : I_Node
VAR
	pNode : POINTER TO Node_F_VN_DivideImages;
END_VAR
pNode := __NEW(Node_F_VN_DivideImages);
Clone := pNode^;
END_METHOD

METHOD PROTECTED OnExecute
hresult.Value := F_VN_DivideImages(
    ipSrcImage1 := ipSrcImage1.Value,
    ipSrcImage2 := ipSrcImage2.Value,
	ipDestImage := ipDestImage.Value,
	hrPrev:= hrPrev.Value);
END_METHOD

METHOD PUBLIC PreExecutionCheck
VAR_INPUT
	Check : I_PreExecutionChecks;
END_VAR
Check.IsTrue(ipSrcImage1.IsValid, 'ipSrcImage1 must contain an image');
Check.IsTrue(ipSrcImage2.IsValid, 'ipSrcImage2 must contain an image');
Check.IsTrue(IsImage1SizeEqualToImage2Size(ipSrcImage1.Value, ipSrcImage2.Value), 'ipSrcImage1 must be the same size as ipSrcImage2');
END_METHOD

END_FUNCTION_BLOCK

// Nodes/Algebraic Image Ops/Node_F_VN_DivideScalarByImage
{attribute 'linkalways'} 
{attribute 'no_explicit_call' := 'This FB is a CLASS and must be accessed using methods or properties'}
{attribute 'enable_dynamic_creation'}
FUNCTION_BLOCK Node_F_VN_DivideScalarByImage EXTENDS VisionNode
VAR
    fScalar : _LREAL(0.0);
    ipSrcImage : _ITcVnImage;
    ipDestImage : _ITcVnImage;
    hrPrev : _HRESULT(S_OK);
	hresult : _HRESULT(S_OK);
END_VAR

METHOD FB_init : BOOL
VAR_INPUT
	bInitRetains : BOOL; // if TRUE, the retain variables are initialized (warm start / cold start)
	bInCopyCode : BOOL;  // if TRUE, the instance afterwards gets moved into the copy code (online change)
END_VAR
AddParameter('fScalar', fScalar);
AddInput('ipSrcImage', ipSrcImage);
AddInput('hrPrev', hrPrev);
AddOutput('ipDestImage', ipDestImage);
AddOutput('hresult',hresult);
END_METHOD

METHOD PUBLIC  Clone : I_Node
VAR
	pNode : POINTER TO Node_F_VN_DivideScalarByImage;
END_VAR
pNode := __NEW(Node_F_VN_DivideScalarByImage);
Clone := pNode^;
END_METHOD

METHOD PROTECTED OnExecute
hresult.Value := F_VN_DivideScalarByImage(
    fScalar := fScalar.Value,
    ipSrcImage := ipSrcImage.Value,
	ipDestImage := ipDestImage.Value,
	hrPrev:= hrPrev.Value);
END_METHOD

METHOD PUBLIC PreExecutionCheck
VAR_INPUT
	Check : I_PreExecutionChecks;
END_VAR
Check.IsTrue(ipSrcImage.IsValid, 'ipSrcImage must contain an image');
END_METHOD

END_FUNCTION_BLOCK

// Nodes/Algebraic Image Ops/Node_F_VN_DivideVectorByImage
{attribute 'linkalways'} 
{attribute 'no_explicit_call' := 'This FB is a CLASS and must be accessed using methods or properties'}
{attribute 'enable_dynamic_creation'}
FUNCTION_BLOCK Node_F_VN_DivideVectorByImage EXTENDS VisionNode
VAR
    aVector : _TcVnVector4_LREAL;
    ipSrcImage : _ITcVnImage;
    ipDestImage : _ITcVnImage;
    hrPrev : _HRESULT(S_OK);
	hresult : _HRESULT(S_OK);
END_VAR

METHOD FB_init : BOOL
VAR_INPUT
	bInitRetains : BOOL; // if TRUE, the retain variables are initialized (warm start / cold start)
	bInCopyCode : BOOL;  // if TRUE, the instance afterwards gets moved into the copy code (online change)
END_VAR
AddInput('aVector', aVector);
AddInput('ipSrcImage', ipSrcImage);
AddInput('hrPrev', hrPrev);
AddOutput('ipDestImage', ipDestImage);
AddOutput('hresult',hresult);
END_METHOD

METHOD PUBLIC  Clone : I_Node
VAR
	pNode : POINTER TO Node_F_VN_DivideVectorByImage;
END_VAR
pNode := __NEW(Node_F_VN_DivideVectorByImage);
Clone := pNode^;
END_METHOD

METHOD PROTECTED OnExecute
hresult.Value := F_VN_DivideVectorByImage(
    aVector := aVector.Value,
    ipSrcImage := ipSrcImage.Value,
	ipDestImage := ipDestImage.Value,
	hrPrev:= hrPrev.Value);
END_METHOD

METHOD PUBLIC PreExecutionCheck
VAR_INPUT
	Check : I_PreExecutionChecks;
END_VAR
Check.IsTrue(ipSrcImage.IsValid, 'ipSrcImage must contain an image');
END_METHOD

END_FUNCTION_BLOCK

// Nodes/Algebraic Image Ops/Node_F_VN_ElementwiseExp
{attribute 'linkalways'} 
{attribute 'no_explicit_call' := 'This FB is a CLASS and must be accessed using methods or properties'}
{attribute 'enable_dynamic_creation'}
FUNCTION_BLOCK Node_F_VN_ElementwiseExp EXTENDS VisionNode
VAR
    ipSrcImage : _ITcVnImage;
    ipDestImage : _ITcVnImage;
    hrPrev : _HRESULT(S_OK);
	hresult : _HRESULT(S_OK);
END_VAR

METHOD FB_init : BOOL
VAR_INPUT
	bInitRetains : BOOL; // if TRUE, the retain variables are initialized (warm start / cold start)
	bInCopyCode : BOOL;  // if TRUE, the instance afterwards gets moved into the copy code (online change)
END_VAR
AddInput('ipSrcImage', ipSrcImage);
AddInput('hrPrev', hrPrev);
AddOutput('ipDestImage', ipDestImage);
AddOutput('hresult',hresult);
END_METHOD

METHOD PUBLIC  Clone : I_Node
VAR
	pNode : POINTER TO Node_F_VN_ElementwiseExp;
END_VAR
pNode := __NEW(Node_F_VN_ElementwiseExp);
Clone := pNode^;
END_METHOD

METHOD PROTECTED OnExecute
hresult.Value := F_VN_ElementwiseExp(
    ipSrcImage := ipSrcImage.Value,
	ipDestImage := ipDestImage.Value,
	hrPrev:= hrPrev.Value);
END_METHOD

METHOD PUBLIC PreExecutionCheck
VAR_INPUT
	Check : I_PreExecutionChecks;
END_VAR
Check.IsTrue(ipSrcImage.IsValid, 'ipSrcImage must contain an image');
Check.IsTrue((ipSrcImage.IsPixelDepth(32) OR
              ipSrcImage.IsPixelDepth(64)), 'ipSrcImage must have 32 or 64 bit pixel depth');
END_METHOD

END_FUNCTION_BLOCK

// Nodes/Algebraic Image Ops/Node_F_VN_ElementwiseLog
{attribute 'linkalways'} 
{attribute 'no_explicit_call' := 'This FB is a CLASS and must be accessed using methods or properties'}
{attribute 'enable_dynamic_creation'}
FUNCTION_BLOCK Node_F_VN_ElementwiseLog EXTENDS VisionNode
VAR
    ipSrcImage : _ITcVnImage;
    ipDestImage : _ITcVnImage;
    hrPrev : _HRESULT(S_OK);
	hresult : _HRESULT(S_OK);
END_VAR

METHOD FB_init : BOOL
VAR_INPUT
	bInitRetains : BOOL; // if TRUE, the retain variables are initialized (warm start / cold start)
	bInCopyCode : BOOL;  // if TRUE, the instance afterwards gets moved into the copy code (online change)
END_VAR
AddInput('ipSrcImage', ipSrcImage);
AddInput('hrPrev', hrPrev);
AddOutput('ipDestImage', ipDestImage);
AddOutput('hresult',hresult);
END_METHOD

METHOD PUBLIC  Clone : I_Node
VAR
	pNode : POINTER TO Node_F_VN_ElementwiseLog;
END_VAR
pNode := __NEW(Node_F_VN_ElementwiseLog);
Clone := pNode^;
END_METHOD

METHOD PROTECTED OnExecute
hresult.Value := F_VN_ElementwiseLog(
    ipSrcImage := ipSrcImage.Value,
	ipDestImage := ipDestImage.Value,
	hrPrev:= hrPrev.Value);
END_METHOD

METHOD PUBLIC PreExecutionCheck
VAR_INPUT
	Check : I_PreExecutionChecks;
END_VAR
Check.IsTrue(ipSrcImage.IsValid, 'ipSrcImage must contain an image');
Check.IsTrue((ipSrcImage.IsPixelDepth(32) OR
              ipSrcImage.IsPixelDepth(64)), 'ipSrcImage must have 32 or 64 bit pixel depth');
END_METHOD

END_FUNCTION_BLOCK

// Nodes/Algebraic Image Ops/Node_F_VN_MaxImage
{attribute 'linkalways'} 
{attribute 'no_explicit_call' := 'This FB is a CLASS and must be accessed using methods or properties'}
{attribute 'enable_dynamic_creation'}
FUNCTION_BLOCK Node_F_VN_MaxImage EXTENDS VisionNode
VAR
    ipSrcImage1 : _ITcVnImage;
    ipSrcImage2 : _ITcVnImage;
    ipDestImage : _ITcVnImage;
    hrPrev : _HRESULT(S_OK);
	hresult : _HRESULT(S_OK);
END_VAR

METHOD FB_init : BOOL
VAR_INPUT
	bInitRetains : BOOL; // if TRUE, the retain variables are initialized (warm start / cold start)
	bInCopyCode : BOOL;  // if TRUE, the instance afterwards gets moved into the copy code (online change)
END_VAR
AddInput('ipSrcImage1', ipSrcImage1);
AddInput('ipSrcImage2', ipSrcImage2);
AddInput('hrPrev', hrPrev);
AddOutput('ipDestImage', ipDestImage);
AddOutput('hresult',hresult);
END_METHOD

METHOD PUBLIC  Clone : I_Node
VAR
	pNode : POINTER TO Node_F_VN_MaxImage;
END_VAR
pNode := __NEW(Node_F_VN_MaxImage);
Clone := pNode^;
END_METHOD

METHOD PROTECTED OnExecute
hresult.Value := F_VN_MaxImage(
    ipSrcImage1 := ipSrcImage1.Value,
    ipSrcImage2 := ipSrcImage2.Value,
	ipDestImage := ipDestImage.Value,
	hrPrev:= hrPrev.Value);
END_METHOD

METHOD PUBLIC PreExecutionCheck
VAR_INPUT
	Check : I_PreExecutionChecks;
END_VAR
Check.IsTrue(ipSrcImage1.IsValid, 'ipSrcImage1 must contain an image');
Check.IsTrue(ipSrcImage2.IsValid, 'ipSrcImage2 must contain an image');
Check.IsTrue(IsImage1SizeEqualToImage2Size(ipSrcImage1.Value, ipSrcImage2.Value), 'ipSrcImage1 must be the same size as ipSrcImage2');
END_METHOD

END_FUNCTION_BLOCK

// Nodes/Algebraic Image Ops/Node_F_VN_MaxImageExp
{attribute 'linkalways'} 
{attribute 'no_explicit_call' := 'This FB is a CLASS and must be accessed using methods or properties'}
{attribute 'enable_dynamic_creation'}
FUNCTION_BLOCK Node_F_VN_MaxImageExp EXTENDS VisionNode
VAR
    ipSrcImage1 : _ITcVnImage;
    ipSrcImage2 : _ITcVnImage;
    ipDestImage : _ITcVnImage;
    ipMask : _ITcVnImage;
    hrPrev : _HRESULT(S_OK);
	hresult : _HRESULT(S_OK);
END_VAR

METHOD FB_init : BOOL
VAR_INPUT
	bInitRetains : BOOL; // if TRUE, the retain variables are initialized (warm start / cold start)
	bInCopyCode : BOOL;  // if TRUE, the instance afterwards gets moved into the copy code (online change)
END_VAR
AddInput('ipSrcImage1', ipSrcImage1);
AddInput('ipSrcImage2', ipSrcImage2);
AddInput('ipMask', ipMask);
AddInput('hrPrev', hrPrev);
AddOutput('ipDestImage', ipDestImage);
AddOutput('hresult',hresult);
END_METHOD

METHOD PUBLIC  Clone : I_Node
VAR
	pNode : POINTER TO Node_F_VN_MaxImageExp;
END_VAR
pNode := __NEW(Node_F_VN_MaxImageExp);
Clone := pNode^;
END_METHOD

METHOD PROTECTED OnExecute
hresult.Value := F_VN_MaxImageExp(
    ipSrcImage1 := ipSrcImage1.Value,
    ipSrcImage2 := ipSrcImage2.Value,
	ipDestImage := ipDestImage.Value,
    ipMask := ipMask.Value,
	hrPrev:= hrPrev.Value);
END_METHOD

METHOD PUBLIC PreExecutionCheck
VAR_INPUT
	Check : I_PreExecutionChecks;
END_VAR
Check.IsTrue(ipSrcImage1.IsValid, 'ipSrcImage1 must contain an image');
Check.IsTrue(ipSrcImage2.IsValid, 'ipSrcImage2 must contain an image');
Check.IsTrue(IsImage1SizeEqualToImage2Size(ipSrcImage1.Value, ipSrcImage2.Value), 'ipSrcImage1 must be the same size as ipSrcImage2');
Check.IsTrue(ipMask.IsValid, 'ipMask must contain an image');
Check.IsTrue(ipMask.HasChannelCount(1), 'ipMask must have 1 channel');
Check.IsTrue(ipMask.IsPixelDepth(8), 'ipMask must have 8 bit pixel depth');
Check.IsTrue(IsImage1SizeEqualToImage2Size(ipMask.Value, ipSrcImage1.Value), 'ipMask must be the same size as ipSrcImage1');
END_METHOD

END_FUNCTION_BLOCK

// Nodes/Algebraic Image Ops/Node_F_VN_MaxImageWithScalar
{attribute 'linkalways'} 
{attribute 'no_explicit_call' := 'This FB is a CLASS and must be accessed using methods or properties'}
{attribute 'enable_dynamic_creation'}
FUNCTION_BLOCK Node_F_VN_MaxImageWithScalar EXTENDS VisionNode
VAR
    fScalar : _LREAL(0.0);
    ipSrcImage : _ITcVnImage;
    ipDestImage : _ITcVnImage;
    hrPrev : _HRESULT(S_OK);
	hresult : _HRESULT(S_OK);
END_VAR

METHOD FB_init : BOOL
VAR_INPUT
	bInitRetains : BOOL; // if TRUE, the retain variables are initialized (warm start / cold start)
	bInCopyCode : BOOL;  // if TRUE, the instance afterwards gets moved into the copy code (online change)
END_VAR
AddParameter('fScalar', fScalar);
AddInput('ipSrcImage', ipSrcImage);
AddInput('hrPrev', hrPrev);
AddOutput('ipDestImage', ipDestImage);
AddOutput('hresult',hresult);
END_METHOD

METHOD PUBLIC  Clone : I_Node
VAR
	pNode : POINTER TO Node_F_VN_MaxImageWithScalar;
END_VAR
pNode := __NEW(Node_F_VN_MaxImageWithScalar);
Clone := pNode^;
END_METHOD

METHOD PROTECTED OnExecute
hresult.Value := F_VN_MaxImageWithScalar(
    fScalar := fScalar.Value,
    ipSrcImage := ipSrcImage.Value,
	ipDestImage := ipDestImage.Value,
	hrPrev:= hrPrev.Value);
END_METHOD

METHOD PUBLIC PreExecutionCheck
VAR_INPUT
	Check : I_PreExecutionChecks;
END_VAR
Check.IsTrue(ipSrcImage.IsValid, 'ipSrcImage must contain an image');
END_METHOD

END_FUNCTION_BLOCK

// Nodes/Algebraic Image Ops/Node_F_VN_MaxImageWithScalarExp
{attribute 'linkalways'} 
{attribute 'no_explicit_call' := 'This FB is a CLASS and must be accessed using methods or properties'}
{attribute 'enable_dynamic_creation'}
FUNCTION_BLOCK Node_F_VN_MaxImageWithScalarExp EXTENDS VisionNode
VAR
    fScalar : _LREAL(0.0);
    ipSrcImage : _ITcVnImage;
    ipDestImage : _ITcVnImage;
    ipMask : _ITcVnImage;
    hrPrev : _HRESULT(S_OK);
	hresult : _HRESULT(S_OK);
END_VAR

METHOD FB_init : BOOL
VAR_INPUT
	bInitRetains : BOOL; // if TRUE, the retain variables are initialized (warm start / cold start)
	bInCopyCode : BOOL;  // if TRUE, the instance afterwards gets moved into the copy code (online change)
END_VAR
AddParameter('fScalar', fScalar);
AddInput('ipSrcImage', ipSrcImage);
AddInput('ipMask', ipMask);
AddInput('hrPrev', hrPrev);
AddOutput('ipDestImage', ipDestImage);
AddOutput('hresult',hresult);
END_METHOD

METHOD PUBLIC  Clone : I_Node
VAR
	pNode : POINTER TO Node_F_VN_MaxImageWithScalarExp;
END_VAR
pNode := __NEW(Node_F_VN_MaxImageWithScalarExp);
Clone := pNode^;
END_METHOD

METHOD PROTECTED OnExecute
hresult.Value := F_VN_MaxImageWithScalarExp(
    fScalar := fScalar.Value,
    ipSrcImage := ipSrcImage.Value,
	ipDestImage := ipDestImage.Value,
    ipMask := ipMask.Value,
	hrPrev:= hrPrev.Value);
END_METHOD

METHOD PUBLIC PreExecutionCheck
VAR_INPUT
	Check : I_PreExecutionChecks;
END_VAR
Check.IsTrue(ipSrcImage.IsValid, 'ipSrcImage must contain an image');
Check.IsTrue(ipMask.IsValid, 'ipMask must contain an image');
Check.IsTrue(ipMask.HasChannelCount(1), 'ipMask must have 1 channel');
Check.IsTrue(ipMask.IsPixelDepth(8), 'ipMask must have 8 bit pixel depth');
Check.IsTrue(IsImage1SizeEqualToImage2Size(ipMask.Value, ipSrcImage.Value), 'ipMask must be the same size as ipSrcImage');
END_METHOD

END_FUNCTION_BLOCK

// Nodes/Algebraic Image Ops/Node_F_VN_MaxImageWithVector
{attribute 'linkalways'} 
{attribute 'no_explicit_call' := 'This FB is a CLASS and must be accessed using methods or properties'}
{attribute 'enable_dynamic_creation'}
FUNCTION_BLOCK Node_F_VN_MaxImageWithVector EXTENDS VisionNode
VAR
    aVector : _TcVnVector4_LREAL;
    ipSrcImage : _ITcVnImage;
    ipDestImage : _ITcVnImage;
    hrPrev : _HRESULT(S_OK);
	hresult : _HRESULT(S_OK);
END_VAR

METHOD FB_init : BOOL
VAR_INPUT
	bInitRetains : BOOL; // if TRUE, the retain variables are initialized (warm start / cold start)
	bInCopyCode : BOOL;  // if TRUE, the instance afterwards gets moved into the copy code (online change)
END_VAR
AddInput('aVector', aVector);
AddInput('ipSrcImage', ipSrcImage);
AddInput('hrPrev', hrPrev);
AddOutput('ipDestImage', ipDestImage);
AddOutput('hresult',hresult);
END_METHOD

METHOD PUBLIC  Clone : I_Node
VAR
	pNode : POINTER TO Node_F_VN_MaxImageWithVector;
END_VAR
pNode := __NEW(Node_F_VN_MaxImageWithVector);
Clone := pNode^;
END_METHOD

METHOD PROTECTED OnExecute
hresult.Value := F_VN_MaxImageWithVector(
    aVector := aVector.Value,
    ipSrcImage := ipSrcImage.Value,
	ipDestImage := ipDestImage.Value,
	hrPrev:= hrPrev.Value);
END_METHOD

METHOD PUBLIC PreExecutionCheck
VAR_INPUT
	Check : I_PreExecutionChecks;
END_VAR
Check.IsTrue(ipSrcImage.IsValid, 'ipSrcImage must contain an image');
END_METHOD

END_FUNCTION_BLOCK

// Nodes/Algebraic Image Ops/Node_F_VN_MaxImageWithVectorExp
{attribute 'linkalways'} 
{attribute 'no_explicit_call' := 'This FB is a CLASS and must be accessed using methods or properties'}
{attribute 'enable_dynamic_creation'}
FUNCTION_BLOCK Node_F_VN_MaxImageWithVectorExp EXTENDS VisionNode
VAR
    aVector : _TcVnVector4_LREAL;
    ipSrcImage : _ITcVnImage;
    ipDestImage : _ITcVnImage;
    ipMask : _ITcVnImage;
    hrPrev : _HRESULT(S_OK);
	hresult : _HRESULT(S_OK);
END_VAR

METHOD FB_init : BOOL
VAR_INPUT
	bInitRetains : BOOL; // if TRUE, the retain variables are initialized (warm start / cold start)
	bInCopyCode : BOOL;  // if TRUE, the instance afterwards gets moved into the copy code (online change)
END_VAR
AddInput('aVector', aVector);
AddInput('ipSrcImage', ipSrcImage);
AddInput('ipMask', ipMask);
AddInput('hrPrev', hrPrev);
AddOutput('ipDestImage', ipDestImage);
AddOutput('hresult',hresult);
END_METHOD

METHOD PUBLIC  Clone : I_Node
VAR
	pNode : POINTER TO Node_F_VN_MaxImageWithVectorExp;
END_VAR
pNode := __NEW(Node_F_VN_MaxImageWithVectorExp);
Clone := pNode^;
END_METHOD

METHOD PROTECTED OnExecute
hresult.Value := F_VN_MaxImageWithVectorExp(
    aVector := aVector.Value,
    ipSrcImage := ipSrcImage.Value,
	ipDestImage := ipDestImage.Value,
    ipMask := ipMask.Value,
	hrPrev:= hrPrev.Value);
END_METHOD

METHOD PUBLIC PreExecutionCheck
VAR_INPUT
	Check : I_PreExecutionChecks;
END_VAR
Check.IsTrue(ipSrcImage.IsValid, 'ipSrcImage must contain an image');
Check.IsTrue(ipMask.IsValid, 'ipMask must contain an image');
Check.IsTrue(ipMask.HasChannelCount(1), 'ipMask must have 1 channel');
Check.IsTrue(ipMask.IsPixelDepth(8), 'ipMask must have 8 bit pixel depth');
Check.IsTrue(IsImage1SizeEqualToImage2Size(ipMask.Value, ipSrcImage.Value), 'ipMask must be the same size as ipSrcImage');
END_METHOD

END_FUNCTION_BLOCK

// Nodes/Algebraic Image Ops/Node_F_VN_MinImage
{attribute 'linkalways'} 
{attribute 'no_explicit_call' := 'This FB is a CLASS and must be accessed using methods or properties'}
{attribute 'enable_dynamic_creation'}
FUNCTION_BLOCK Node_F_VN_MinImage EXTENDS VisionNode
VAR
    ipSrcImage1 : _ITcVnImage;
    ipSrcImage2 : _ITcVnImage;
    ipDestImage : _ITcVnImage;
    hrPrev : _HRESULT(S_OK);
	hresult : _HRESULT(S_OK);
END_VAR

METHOD FB_init : BOOL
VAR_INPUT
	bInitRetains : BOOL; // if TRUE, the retain variables are initialized (warm start / cold start)
	bInCopyCode : BOOL;  // if TRUE, the instance afterwards gets moved into the copy code (online change)
END_VAR
AddInput('ipSrcImage1', ipSrcImage1);
AddInput('ipSrcImage2', ipSrcImage2);
AddInput('hrPrev', hrPrev);
AddOutput('ipDestImage', ipDestImage);
AddOutput('hresult',hresult);
END_METHOD

METHOD PUBLIC  Clone : I_Node
VAR
	pNode : POINTER TO Node_F_VN_MinImage;
END_VAR
pNode := __NEW(Node_F_VN_MinImage);
Clone := pNode^;
END_METHOD

METHOD PROTECTED OnExecute
hresult.Value := F_VN_MinImage(
    ipSrcImage1 := ipSrcImage1.Value,
    ipSrcImage2 := ipSrcImage2.Value,
	ipDestImage := ipDestImage.Value,
	hrPrev:= hrPrev.Value);
END_METHOD

METHOD PUBLIC PreExecutionCheck
VAR_INPUT
	Check : I_PreExecutionChecks;
END_VAR
Check.IsTrue(ipSrcImage1.IsValid, 'ipSrcImage1 must contain an image');
Check.IsTrue(ipSrcImage2.IsValid, 'ipSrcImage2 must contain an image');
Check.IsTrue(IsImage1SizeEqualToImage2Size(ipSrcImage1.Value, ipSrcImage2.Value), 'ipSrcImage1 must be the same size as ipSrcImage2');
END_METHOD

END_FUNCTION_BLOCK

// Nodes/Algebraic Image Ops/Node_F_VN_MinImageExp
{attribute 'linkalways'} 
{attribute 'no_explicit_call' := 'This FB is a CLASS and must be accessed using methods or properties'}
{attribute 'enable_dynamic_creation'}
FUNCTION_BLOCK Node_F_VN_MinImageExp EXTENDS VisionNode
VAR
    ipSrcImage1 : _ITcVnImage;
    ipSrcImage2 : _ITcVnImage;
    ipDestImage : _ITcVnImage;
    ipMask : _ITcVnImage;
    hrPrev : _HRESULT(S_OK);
	hresult : _HRESULT(S_OK);
END_VAR

METHOD FB_init : BOOL
VAR_INPUT
	bInitRetains : BOOL; // if TRUE, the retain variables are initialized (warm start / cold start)
	bInCopyCode : BOOL;  // if TRUE, the instance afterwards gets moved into the copy code (online change)
END_VAR
AddInput('ipSrcImage1', ipSrcImage1);
AddInput('ipSrcImage2', ipSrcImage2);
AddInput('ipMask', ipMask);
AddInput('hrPrev', hrPrev);
AddOutput('ipDestImage', ipDestImage);
AddOutput('hresult',hresult);
END_METHOD

METHOD PUBLIC  Clone : I_Node
VAR
	pNode : POINTER TO Node_F_VN_MinImageExp;
END_VAR
pNode := __NEW(Node_F_VN_MinImageExp);
Clone := pNode^;
END_METHOD

METHOD PROTECTED OnExecute
hresult.Value := F_VN_MinImageExp(
    ipSrcImage1 := ipSrcImage1.Value,
    ipSrcImage2 := ipSrcImage2.Value,
	ipDestImage := ipDestImage.Value,
    ipMask := ipMask.Value,
	hrPrev:= hrPrev.Value);
END_METHOD

METHOD PUBLIC PreExecutionCheck
VAR_INPUT
	Check : I_PreExecutionChecks;
END_VAR
Check.IsTrue(ipSrcImage1.IsValid, 'ipSrcImage1 must contain an image');
Check.IsTrue(ipSrcImage2.IsValid, 'ipSrcImage2 must contain an image');
Check.IsTrue(IsImage1SizeEqualToImage2Size(ipSrcImage1.Value, ipSrcImage2.Value), 'ipSrcImage1 must be the same size as ipSrcImage2');
Check.IsTrue(ipMask.IsValid, 'ipMask must contain an image');
Check.IsTrue(ipMask.HasChannelCount(1), 'ipMask must have 1 channel');
Check.IsTrue(ipMask.IsPixelDepth(8), 'ipMask must have 8 bit pixel depth');
Check.IsTrue(IsImage1SizeEqualToImage2Size(ipMask.Value, ipSrcImage1.Value), 'ipMask must be the same size as ipSrcImage1');
END_METHOD

END_FUNCTION_BLOCK

// Nodes/Algebraic Image Ops/Node_F_VN_MinImageWithScalar
{attribute 'linkalways'} 
{attribute 'no_explicit_call' := 'This FB is a CLASS and must be accessed using methods or properties'}
{attribute 'enable_dynamic_creation'}
FUNCTION_BLOCK Node_F_VN_MinImageWithScalar EXTENDS VisionNode
VAR
    fScalar : _LREAL(0.0);
    ipSrcImage : _ITcVnImage;
    ipDestImage : _ITcVnImage;
    hrPrev : _HRESULT(S_OK);
	hresult : _HRESULT(S_OK);
END_VAR

METHOD FB_init : BOOL
VAR_INPUT
	bInitRetains : BOOL; // if TRUE, the retain variables are initialized (warm start / cold start)
	bInCopyCode : BOOL;  // if TRUE, the instance afterwards gets moved into the copy code (online change)
END_VAR
AddParameter('fScalar', fScalar);
AddInput('ipSrcImage', ipSrcImage);
AddInput('hrPrev', hrPrev);
AddOutput('ipDestImage', ipDestImage);
AddOutput('hresult',hresult);
END_METHOD

METHOD PUBLIC  Clone : I_Node
VAR
	pNode : POINTER TO Node_F_VN_MinImageWithScalar;
END_VAR
pNode := __NEW(Node_F_VN_MinImageWithScalar);
Clone := pNode^;
END_METHOD

METHOD PROTECTED OnExecute
hresult.Value := F_VN_MinImageWithScalar(
    fScalar := fScalar.Value,
    ipSrcImage := ipSrcImage.Value,
	ipDestImage := ipDestImage.Value,
	hrPrev:= hrPrev.Value);
END_METHOD

METHOD PUBLIC PreExecutionCheck
VAR_INPUT
	Check : I_PreExecutionChecks;
END_VAR
Check.IsTrue(ipSrcImage.IsValid, 'ipSrcImage must contain an image');
END_METHOD

END_FUNCTION_BLOCK

// Nodes/Algebraic Image Ops/Node_F_VN_MinImageWithScalarExp
{attribute 'linkalways'} 
{attribute 'no_explicit_call' := 'This FB is a CLASS and must be accessed using methods or properties'}
{attribute 'enable_dynamic_creation'}
FUNCTION_BLOCK Node_F_VN_MinImageWithScalarExp EXTENDS VisionNode
VAR
    fScalar : _LREAL(0.0);
    ipSrcImage : _ITcVnImage;
    ipDestImage : _ITcVnImage;
    ipMask : _ITcVnImage;
    hrPrev : _HRESULT(S_OK);
	hresult : _HRESULT(S_OK);
END_VAR

METHOD FB_init : BOOL
VAR_INPUT
	bInitRetains : BOOL; // if TRUE, the retain variables are initialized (warm start / cold start)
	bInCopyCode : BOOL;  // if TRUE, the instance afterwards gets moved into the copy code (online change)
END_VAR
AddParameter('fScalar', fScalar);
AddInput('ipSrcImage', ipSrcImage);
AddInput('ipMask', ipMask);
AddInput('hrPrev', hrPrev);
AddOutput('ipDestImage', ipDestImage);
AddOutput('hresult',hresult);
END_METHOD

METHOD PUBLIC  Clone : I_Node
VAR
	pNode : POINTER TO Node_F_VN_MinImageWithScalarExp;
END_VAR
pNode := __NEW(Node_F_VN_MinImageWithScalarExp);
Clone := pNode^;
END_METHOD

METHOD PROTECTED OnExecute
hresult.Value := F_VN_MinImageWithScalarExp(
    fScalar := fScalar.Value,
    ipSrcImage := ipSrcImage.Value,
	ipDestImage := ipDestImage.Value,
    ipMask := ipMask.Value,
	hrPrev:= hrPrev.Value);
END_METHOD

METHOD PUBLIC PreExecutionCheck
VAR_INPUT
	Check : I_PreExecutionChecks;
END_VAR
Check.IsTrue(ipSrcImage.IsValid, 'ipSrcImage must contain an image');
Check.IsTrue(ipMask.IsValid, 'ipMask must contain an image');
Check.IsTrue(ipMask.HasChannelCount(1), 'ipMask must have 1 channel');
Check.IsTrue(ipMask.IsPixelDepth(8), 'ipMask must have 8 bit pixel depth');
Check.IsTrue(IsImage1SizeEqualToImage2Size(ipMask.Value, ipSrcImage.Value), 'ipMask must be the same size as ipSrcImage');
END_METHOD

END_FUNCTION_BLOCK

// Nodes/Algebraic Image Ops/Node_F_VN_MinImageWithVector
{attribute 'linkalways'} 
{attribute 'no_explicit_call' := 'This FB is a CLASS and must be accessed using methods or properties'}
{attribute 'enable_dynamic_creation'}
FUNCTION_BLOCK Node_F_VN_MinImageWithVector EXTENDS VisionNode
VAR
    aVector : _TcVnVector4_LREAL;
    ipSrcImage : _ITcVnImage;
    ipDestImage : _ITcVnImage;
    hrPrev : _HRESULT(S_OK);
	hresult : _HRESULT(S_OK);
END_VAR

METHOD FB_init : BOOL
VAR_INPUT
	bInitRetains : BOOL; // if TRUE, the retain variables are initialized (warm start / cold start)
	bInCopyCode : BOOL;  // if TRUE, the instance afterwards gets moved into the copy code (online change)
END_VAR
AddInput('aVector', aVector);
AddInput('ipSrcImage', ipSrcImage);
AddInput('hrPrev', hrPrev);
AddOutput('ipDestImage', ipDestImage);
AddOutput('hresult',hresult);
END_METHOD

METHOD PUBLIC  Clone : I_Node
VAR
	pNode : POINTER TO Node_F_VN_MinImageWithVector;
END_VAR
pNode := __NEW(Node_F_VN_MinImageWithVector);
Clone := pNode^;
END_METHOD

METHOD PROTECTED OnExecute
hresult.Value := F_VN_MinImageWithVector(
    aVector := aVector.Value,
    ipSrcImage := ipSrcImage.Value,
	ipDestImage := ipDestImage.Value,
	hrPrev:= hrPrev.Value);
END_METHOD

METHOD PUBLIC PreExecutionCheck
VAR_INPUT
	Check : I_PreExecutionChecks;
END_VAR
Check.IsTrue(ipSrcImage.IsValid, 'ipSrcImage must contain an image');
END_METHOD

END_FUNCTION_BLOCK

// Nodes/Algebraic Image Ops/Node_F_VN_MinImageWithVectorExp
{attribute 'linkalways'} 
{attribute 'no_explicit_call' := 'This FB is a CLASS and must be accessed using methods or properties'}
{attribute 'enable_dynamic_creation'}
FUNCTION_BLOCK Node_F_VN_MinImageWithVectorExp EXTENDS VisionNode
VAR
    aVector : _TcVnVector4_LREAL;
    ipSrcImage : _ITcVnImage;
    ipDestImage : _ITcVnImage;
    ipMask : _ITcVnImage;
    hrPrev : _HRESULT(S_OK);
	hresult : _HRESULT(S_OK);
END_VAR

METHOD FB_init : BOOL
VAR_INPUT
	bInitRetains : BOOL; // if TRUE, the retain variables are initialized (warm start / cold start)
	bInCopyCode : BOOL;  // if TRUE, the instance afterwards gets moved into the copy code (online change)
END_VAR
AddInput('aVector', aVector);
AddInput('ipSrcImage', ipSrcImage);
AddInput('ipMask', ipMask);
AddInput('hrPrev', hrPrev);
AddOutput('ipDestImage', ipDestImage);
AddOutput('hresult',hresult);
END_METHOD

METHOD PUBLIC  Clone : I_Node
VAR
	pNode : POINTER TO Node_F_VN_MinImageWithVectorExp;
END_VAR
pNode := __NEW(Node_F_VN_MinImageWithVectorExp);
Clone := pNode^;
END_METHOD

METHOD PROTECTED OnExecute
hresult.Value := F_VN_MinImageWithVectorExp(
    aVector := aVector.Value,
    ipSrcImage := ipSrcImage.Value,
	ipDestImage := ipDestImage.Value,
    ipMask := ipMask.Value,
	hrPrev:= hrPrev.Value);
END_METHOD

METHOD PUBLIC PreExecutionCheck
VAR_INPUT
	Check : I_PreExecutionChecks;
END_VAR
Check.IsTrue(ipSrcImage.IsValid, 'ipSrcImage must contain an image');
Check.IsTrue(ipMask.IsValid, 'ipMask must contain an image');
Check.IsTrue(ipMask.HasChannelCount(1), 'ipMask must have 1 channel');
Check.IsTrue(ipMask.IsPixelDepth(8), 'ipMask must have 8 bit pixel depth');
Check.IsTrue(IsImage1SizeEqualToImage2Size(ipMask.Value, ipSrcImage.Value), 'ipMask must be the same size as ipSrcImage');
END_METHOD

END_FUNCTION_BLOCK

// Nodes/Algebraic Image Ops/Node_F_VN_MultiplyImages
{attribute 'linkalways'} 
{attribute 'no_explicit_call' := 'This FB is a CLASS and must be accessed using methods or properties'}
{attribute 'enable_dynamic_creation'}
FUNCTION_BLOCK Node_F_VN_MultiplyImages EXTENDS VisionNode
VAR
    ipSrcImage1 : _ITcVnImage;
    ipSrcImage2 : _ITcVnImage;
    ipDestImage : _ITcVnImage;
    hrPrev : _HRESULT(S_OK);
	hresult : _HRESULT(S_OK);
END_VAR

METHOD FB_init : BOOL
VAR_INPUT
	bInitRetains : BOOL; // if TRUE, the retain variables are initialized (warm start / cold start)
	bInCopyCode : BOOL;  // if TRUE, the instance afterwards gets moved into the copy code (online change)
END_VAR
AddInput('ipSrcImage1', ipSrcImage1);
AddInput('ipSrcImage2', ipSrcImage2);
AddInput('hrPrev', hrPrev);
AddOutput('ipDestImage', ipDestImage);
AddOutput('hresult',hresult);
END_METHOD

METHOD PUBLIC  Clone : I_Node
VAR
	pNode : POINTER TO Node_F_VN_MultiplyImages;
END_VAR
pNode := __NEW(Node_F_VN_MultiplyImages);
Clone := pNode^;
END_METHOD

METHOD PROTECTED OnExecute
hresult.Value := F_VN_MultiplyImages(
    ipSrcImage1 := ipSrcImage1.Value,
    ipSrcImage2 := ipSrcImage2.Value,
	ipDestImage := ipDestImage.Value,
	hrPrev:= hrPrev.Value);
END_METHOD

METHOD PUBLIC PreExecutionCheck
VAR_INPUT
	Check : I_PreExecutionChecks;
END_VAR
Check.IsTrue(ipSrcImage1.IsValid, 'ipSrcImage1 must contain an image');
Check.IsTrue(ipSrcImage2.IsValid, 'ipSrcImage2 must contain an image');
Check.IsTrue(IsImage1SizeEqualToImage2Size(ipSrcImage1.Value, ipSrcImage2.Value), 'ipSrcImage1 must be the same size as ipSrcImage2');
END_METHOD

END_FUNCTION_BLOCK

// Nodes/Algebraic Image Ops/Node_F_VN_MultiplyImageWithScalar
{attribute 'linkalways'} 
{attribute 'no_explicit_call' := 'This FB is a CLASS and must be accessed using methods or properties'}
{attribute 'enable_dynamic_creation'}
FUNCTION_BLOCK Node_F_VN_MultiplyImageWithScalar EXTENDS VisionNode
VAR
    fScalar : _LREAL(0.0);
    ipSrcImage : _ITcVnImage;
    ipDestImage : _ITcVnImage;
    hrPrev : _HRESULT(S_OK);
	hresult : _HRESULT(S_OK);
END_VAR

METHOD FB_init : BOOL
VAR_INPUT
	bInitRetains : BOOL; // if TRUE, the retain variables are initialized (warm start / cold start)
	bInCopyCode : BOOL;  // if TRUE, the instance afterwards gets moved into the copy code (online change)
END_VAR
AddParameter('fScalar', fScalar);
AddInput('ipSrcImage', ipSrcImage);
AddInput('hrPrev', hrPrev);
AddOutput('ipDestImage', ipDestImage);
AddOutput('hresult',hresult);
END_METHOD

METHOD PUBLIC  Clone : I_Node
VAR
	pNode : POINTER TO Node_F_VN_MultiplyImageWithScalar;
END_VAR
pNode := __NEW(Node_F_VN_MultiplyImageWithScalar);
Clone := pNode^;
END_METHOD

METHOD PROTECTED OnExecute
hresult.Value := F_VN_MultiplyImageWithScalar(
    fScalar := fScalar.Value,
    ipSrcImage := ipSrcImage.Value,
	ipDestImage := ipDestImage.Value,
	hrPrev:= hrPrev.Value);
END_METHOD

METHOD PUBLIC PreExecutionCheck
VAR_INPUT
	Check : I_PreExecutionChecks;
END_VAR
Check.IsTrue(ipSrcImage.IsValid, 'ipSrcImage must contain an image');
END_METHOD

END_FUNCTION_BLOCK

// Nodes/Algebraic Image Ops/Node_F_VN_MultiplyImageWithVector
{attribute 'linkalways'} 
{attribute 'no_explicit_call' := 'This FB is a CLASS and must be accessed using methods or properties'}
{attribute 'enable_dynamic_creation'}
FUNCTION_BLOCK Node_F_VN_MultiplyImageWithVector EXTENDS VisionNode
VAR
    aVector : _TcVnVector4_LREAL;
    ipSrcImage : _ITcVnImage;
    ipDestImage : _ITcVnImage;
    hrPrev : _HRESULT(S_OK);
	hresult : _HRESULT(S_OK);
END_VAR

METHOD FB_init : BOOL
VAR_INPUT
	bInitRetains : BOOL; // if TRUE, the retain variables are initialized (warm start / cold start)
	bInCopyCode : BOOL;  // if TRUE, the instance afterwards gets moved into the copy code (online change)
END_VAR
AddInput('aVector', aVector);
AddInput('ipSrcImage', ipSrcImage);
AddInput('hrPrev', hrPrev);
AddOutput('ipDestImage', ipDestImage);
AddOutput('hresult',hresult);
END_METHOD

METHOD PUBLIC  Clone : I_Node
VAR
	pNode : POINTER TO Node_F_VN_MultiplyImageWithVector;
END_VAR
pNode := __NEW(Node_F_VN_MultiplyImageWithVector);
Clone := pNode^;
END_METHOD

METHOD PROTECTED OnExecute
hresult.Value := F_VN_MultiplyImageWithVector(
    aVector := aVector.Value,
    ipSrcImage := ipSrcImage.Value,
	ipDestImage := ipDestImage.Value,
	hrPrev:= hrPrev.Value);
END_METHOD

METHOD PUBLIC PreExecutionCheck
VAR_INPUT
	Check : I_PreExecutionChecks;
END_VAR
Check.IsTrue(ipSrcImage.IsValid, 'ipSrcImage must contain an image');
END_METHOD

END_FUNCTION_BLOCK

// Nodes/Algebraic Image Ops/Node_F_VN_SubtractImageFromScalar
{attribute 'linkalways'} 
{attribute 'no_explicit_call' := 'This FB is a CLASS and must be accessed using methods or properties'}
{attribute 'enable_dynamic_creation'}
FUNCTION_BLOCK Node_F_VN_SubtractImageFromScalar EXTENDS VisionNode
VAR
    fScalar : _LREAL(0.0);
    ipSrcImage : _ITcVnImage;
    ipDestImage : _ITcVnImage;
    hrPrev : _HRESULT(S_OK);
	hresult : _HRESULT(S_OK);
END_VAR

METHOD FB_init : BOOL
VAR_INPUT
	bInitRetains : BOOL; // if TRUE, the retain variables are initialized (warm start / cold start)
	bInCopyCode : BOOL;  // if TRUE, the instance afterwards gets moved into the copy code (online change)
END_VAR
AddParameter('fScalar', fScalar);
AddInput('ipSrcImage', ipSrcImage);
AddInput('hrPrev', hrPrev);
AddOutput('ipDestImage', ipDestImage);
AddOutput('hresult',hresult);
END_METHOD

METHOD PUBLIC  Clone : I_Node
VAR
	pNode : POINTER TO Node_F_VN_SubtractImageFromScalar;
END_VAR
pNode := __NEW(Node_F_VN_SubtractImageFromScalar);
Clone := pNode^;
END_METHOD

